// Functions/Keypoint Features/F_VN_FindReferenceKeyPointsInImageAKAZE

	{attribute 'TcIecLibraryType'}
	{attribute 'external_name' := 'F_VN_FindReferenceKeyPointsInImageAKAZE_GUID_B9801059_E7E5_45E6_F0CA_70766AD6A2AB'}
	(* Searches a reference image, represented by its AKAZE keypoints and corresponding descriptors, in a given source image (uses the default TcVnParamsAKAZE parameters). *)
	FUNCTION F_VN_FindReferenceKeyPointsInImageAKAZE : HRESULT
	VAR_INPUT
		ipSrcImage	:	ITcVnImage;	(* Source image *)
		ipRefKeyPoints	:	ITcVnContainer;	(* KeyPoints of the reference image, e.g. computed with F_VN_KeyPointsAndDescriptorsAKAZE (ContainerType_Vector_TcVnKeyPoint) *)
		ipRefDescriptors	:	ITcVnImage;	(* Descriptors of the reference image KeyPoints, e.g. computed with F_VN_KeyPointsAndDescriptorsAKAZE *)
		nRefImageWidth	:	UDINT;	(* Width of the reference image in pixels *)
		nRefImageHeight	:	UDINT;	(* Height of the reference image in pixels *)
		ipEdgePoints	:	REFERENCE TO ITcVnContainer;	(* Returns a container with the 4 edge points of the reference image transformed into ipSrcImage coordinates (ContainerType_Vector_TcVnPoint2_REAL) *)
		fMaxDist	:	REAL;	(* Maximum allowed descriptor distance (-1 disables this filter criterion) *)
		fMaxKnnRatio	:	REAL;	(* Maximum allowed distance ratio between first and second best match ([0..1], -1 disables this filter criterion) *)
		hrPrev	:	HRESULT;	(* HRESULT indicating the result of previous operations (If SUCCEEDED(hrPrev) equals false, no operation is executed.) *)
	END_VAR
	VAR_OUTPUT
		aPerspectiveTransform	:	TcVnMatrix3x3_LREAL;	(* Returns the perspective transformation matrix, which transforms the reference points to the source points *)
		nNumberOfGoodMatches	:	UDINT;	(* Return the number of good matches *)
		nNumberOfInliers	:	UDINT;	(* Return the number of inlier matches *)
	END_VAR

END_FUNCTION

// Functions/Keypoint Features/F_VN_KeyPointsAndDescriptorsAKAZE

	{attribute 'TcIecLibraryType'}
	{attribute 'external_name' := 'F_VN_KeyPointsAndDescriptorsAKAZE_GUID_33FCE752_CC73_4619_CE24_ACBC29908D23'}
	(* Detects keypoints and compute descriptors using the AKAZE method. *)
	FUNCTION F_VN_KeyPointsAndDescriptorsAKAZE : HRESULT
	VAR_INPUT
		ipSrcImage	:	ITcVnImage;	(* Source image *)
		ipKeyPoints	:	REFERENCE TO ITcVnContainer;	(* Returns a container which is filled with the keypoints (ContainerType_Vector_TcVnKeyPoint; Non-zero interface pointers are reused.) *)
		ipDescriptors	:	REFERENCE TO ITcVnImage;	(* Descriptor image (set to 0 if not required; 1 descriptor in each row; An appropriate image will be created if required.) *)
		hrPrev	:	HRESULT;	(* HRESULT indicating the result of previous operations (If SUCCEEDED(hrPrev) equals false, no operation is executed.) *)
	END_VAR

END_FUNCTION

// Functions/Keypoint Features/F_VN_FindReferenceKeyPointsInImageAKAZEExp

	{attribute 'TcIecLibraryType'}
	{attribute 'external_name' := 'F_VN_FindReferenceKeyPointsInImageAKAZEExp_GUID_5A20AA7D_A742_4EBE_E505_E1E5875E6765'}
	(* Searches a reference image, represented by its AKAZE keypoints and corresponding descriptors, in a given source image. (expert function) *)
	FUNCTION F_VN_FindReferenceKeyPointsInImageAKAZEExp : HRESULT
	VAR_INPUT
		ipSrcImage	:	ITcVnImage;	(* Source image *)
		ipRefKeyPoints	:	ITcVnContainer;	(* KeyPoints of the reference image, e.g. computed with F_VN_KeyPointsAndDescriptorsAKAZE (ContainerType_Vector_TcVnKeyPoint) *)
		ipRefDescriptors	:	ITcVnImage;	(* Descriptors of the reference image KeyPoints, e.g. computed with F_VN_KeyPointsAndDescriptorsAKAZE *)
		nRefImageWidth	:	UDINT;	(* Width of the reference image in pixels *)
		nRefImageHeight	:	UDINT;	(* Height of the reference image in pixels *)
		ipEdgePoints	:	REFERENCE TO ITcVnContainer;	(* Returns a container with the 4 edge points of the reference image transformed into ipSrcImage coordinates (ContainerType_Vector_TcVnPoint2_REAL) *)
		fMaxDist	:	REAL;	(* Maximum allowed descriptor distance (-1 disables this filter criterion) *)
		fMaxKnnRatio	:	REAL;	(* Maximum allowed distance ratio between first and second best match ([0..1], -1 disables this filter criterion) *)
		eNormType	:	ETcVnNormalizationType;	(* Normalization type used for descriptor matching *)
		ipSrcImageMask	:	ITcVnImage;	(* Mask to specify, where to look for keypoints in ipSrcImage (set to 0 if no mask required) *)
	END_VAR
	VAR_IN_OUT
		stAkazeParams	:	TcVnParamsAKAZE;	(* Parameters to configure the keypoint and descriptor computation for ipSrcImage (resulting descriptors must be compatible to ipRefDescriptors!) *)
	END_VAR
	VAR_INPUT
		eAlgorithm	:	ETcVnEstimationAlgorithm;	(* Estimation algorithm used for computing the perspective transformation between the two point sets *)
		fReprojThreshold	:	LREAL;	(* Maximum allowed reprojection error to treat a point pair as an inlier (only used if eAlgorithm is RANSAC, RHO) *)
		nMaxIterations	:	UDINT;	(* Maximum number of RANSAC iterations *)
		fConfidence	:	LREAL;	(* Confidence (0..1) *)
		hrPrev	:	HRESULT;	(* HRESULT indicating the result of previous operations (If SUCCEEDED(hrPrev) equals false, no operation is executed.) *)
	END_VAR
	VAR_OUTPUT
		aPerspectiveTransform	:	TcVnMatrix3x3_LREAL;	(* Returns the perspective transformation matrix, which transforms the reference points to the source points  *)
		nNumberOfGoodMatches	:	UDINT;	(* Return the number of good matches *)
		nNumberOfInliers	:	UDINT;	(* Return the number of inlier matches *)
	END_VAR

END_FUNCTION

// Functions/Keypoint Features/F_VN_FindReferenceKeyPointsInImageBRISK

	{attribute 'TcIecLibraryType'}
	{attribute 'external_name' := 'F_VN_FindReferenceKeyPointsInImageBRISK_GUID_C6B47D52_F5A1_4A13_CF78_EFB52692276F'}
	(* Searches a reference image, represented by its BRISK keypoints and corresponding descriptors, in a given source image (uses the default TcVnParamsBRISK parameters). *)
	FUNCTION F_VN_FindReferenceKeyPointsInImageBRISK : HRESULT
	VAR_INPUT
		ipSrcImage	:	ITcVnImage;	(* Source image *)
		ipRefKeyPoints	:	ITcVnContainer;	(* KeyPoints of the reference image, e.g. computed with F_VN_KeyPointsAndDescriptorsBRISK (ContainerType_Vector_TcVnKeyPoint) *)
		ipRefDescriptors	:	ITcVnImage;	(* Descriptors of the reference image KeyPoints, e.g. computed with F_VN_KeyPointsAndDescriptorsBRISK *)
		nRefImageWidth	:	UDINT;	(* Width of the reference image in pixels *)
		nRefImageHeight	:	UDINT;	(* Height of the reference image in pixels *)
		ipEdgePoints	:	REFERENCE TO ITcVnContainer;	(* Returns a container with the 4 edge points of the reference image transformed into ipSrcImage coordinates (ContainerType_Vector_TcVnPoint2_REAL) *)
		fMaxDist	:	REAL;	(* Maximum allowed descriptor distance (-1 disables this filter criterion) *)
		fMaxKnnRatio	:	REAL;	(* Maximum allowed distance ratio between first and second best match ([0..1], -1 disables this filter criterion) *)
		hrPrev	:	HRESULT;	(* HRESULT indicating the result of previous operations (If SUCCEEDED(hrPrev) equals false, no operation is executed.) *)
	END_VAR
	VAR_OUTPUT
		aPerspectiveTransform	:	TcVnMatrix3x3_LREAL;	(* Returns the perspective transformation matrix, which transforms the reference points to the source points  *)
		nNumberOfGoodMatches	:	UDINT;	(* Return the number of good matches *)
		nNumberOfInliers	:	UDINT;	(* Return the number of inlier matches *)
	END_VAR

END_FUNCTION

// Functions/Keypoint Features/F_VN_KeyPointsAndDescriptorsBRISK

	{attribute 'TcIecLibraryType'}
	{attribute 'external_name' := 'F_VN_KeyPointsAndDescriptorsBRISK_GUID_84C0A1DE_69BD_404B_FE31_2FE04FC65E23'}
	(* Detects keypoints and compute descriptors using the BRISK method. *)
	FUNCTION F_VN_KeyPointsAndDescriptorsBRISK : HRESULT
	VAR_INPUT
		ipSrcImage	:	ITcVnImage;	(* Source image *)
		ipKeyPoints	:	REFERENCE TO ITcVnContainer;	(* Returns a container which is filled with the keypoints (ContainerType_Vector_TcVnKeyPoint; Non-zero interface pointers are reused.) *)
		ipDescriptors	:	REFERENCE TO ITcVnImage;	(* Descriptor image (set to 0 if not required; 1 descriptor in each row; An appropriate image will be created if required.) *)
		hrPrev	:	HRESULT;	(* HRESULT indicating the result of previous operations (If SUCCEEDED(hrPrev) equals false, no operation is executed.) *)
	END_VAR

END_FUNCTION

// Functions/Keypoint Features/F_VN_FindReferenceKeyPointsInImageBRISKExp

	{attribute 'TcIecLibraryType'}
	{attribute 'external_name' := 'F_VN_FindReferenceKeyPointsInImageBRISKExp_GUID_84B8D030_BDDF_4ECF_E2AC_C4FA02ED163C'}
	(* Searches a reference image, represented by its BRISK keypoints and corresponding descriptors, in a given source image. (expert function) *)
	FUNCTION F_VN_FindReferenceKeyPointsInImageBRISKExp : HRESULT
	VAR_INPUT
		ipSrcImage	:	ITcVnImage;	(* Source image *)
		ipRefKeyPoints	:	ITcVnContainer;	(* KeyPoints of the reference image, e.g. computed with F_VN_KeyPointsAndDescriptorsBRISK (ContainerType_Vector_TcVnKeyPoint) *)
		ipRefDescriptors	:	ITcVnImage;	(* Descriptors of the reference image KeyPoints, e.g. computed with F_VN_KeyPointsAndDescriptorsBRISK *)
		nRefImageWidth	:	UDINT;	(* Width of the reference image in pixels *)
		nRefImageHeight	:	UDINT;	(* Height of the reference image in pixels *)
		ipEdgePoints	:	REFERENCE TO ITcVnContainer;	(* Returns a container with the 4 edge points of the reference image transformed into ipSrcImage coordinates (ContainerType_Vector_TcVnPoint2_REAL) *)
		fMaxDist	:	REAL;	(* Maximum allowed descriptor distance (-1 disables this filter criterion) *)
		fMaxKnnRatio	:	REAL;	(* Maximum allowed distance ratio between first and second best match ([0..1], -1 disables this filter criterion) *)
		eNormType	:	ETcVnNormalizationType;	(* Normalization type used for descriptor matching *)
		ipSrcImageMask	:	ITcVnImage;	(* Mask to specify, where to look for keypoints in ipSrcImage (set to 0 if no mask required) *)
	END_VAR
	VAR_IN_OUT
		stBriskParams	:	TcVnParamsBRISK;	(* Parameters to configure the keypoint and descriptor computation for ipSrcImage (resulting descriptors must be compatible to ipRefDescriptors!) *)
	END_VAR
	VAR_INPUT
		eAlgorithm	:	ETcVnEstimationAlgorithm;	(* Estimation algorithm used for computing the perspective transformation between the two point sets *)
		fReprojThreshold	:	LREAL;	(* Maximum allowed reprojection error to treat a point pair as an inlier (only used if eAlgorithm is RANSAC, RHO) *)
		nMaxIterations	:	UDINT;	(* Maximum number of RANSAC iterations *)
		fConfidence	:	LREAL;	(* Confidence (0..1) *)
		hrPrev	:	HRESULT;	(* HRESULT indicating the result of previous operations (If SUCCEEDED(hrPrev) equals false, no operation is executed.) *)
	END_VAR
	VAR_OUTPUT
		aPerspectiveTransform	:	TcVnMatrix3x3_LREAL;	(* Returns the perspective transformation matrix, which transforms the reference points to the source points  *)
		nNumberOfGoodMatches	:	UDINT;	(* Return the number of good matches *)
		nNumberOfInliers	:	UDINT;	(* Return the number of inlier matches *)
	END_VAR

END_FUNCTION

// Functions/Keypoint Features/F_VN_FindReferenceKeyPointsInImageORB

	{attribute 'TcIecLibraryType'}
	{attribute 'external_name' := 'F_VN_FindReferenceKeyPointsInImageORB_GUID_A7F5A2C2_C6E4_44AD_C84D_FFDC882441D3'}
	(* Searches a reference image, represented by its ORB keypoints and corresponding descriptors, in a given source image (uses the default TcVnParamsORB parameters). *)
	FUNCTION F_VN_FindReferenceKeyPointsInImageORB : HRESULT
	VAR_INPUT
		ipSrcImage	:	ITcVnImage;	(* Source image *)
		ipRefKeyPoints	:	ITcVnContainer;	(* KeyPoints of the reference image, e.g. computed with F_VN_KeyPointsAndDescriptorsORB (ContainerType_Vector_TcVnKeyPoint) *)
		ipRefDescriptors	:	ITcVnImage;	(* Descriptors of the reference image KeyPoints, e.g. computed with F_VN_KeyPointsAndDescriptorsORB *)
		nRefImageWidth	:	UDINT;	(* Width of the reference image in pixels *)
		nRefImageHeight	:	UDINT;	(* Height of the reference image in pixels *)
		ipEdgePoints	:	REFERENCE TO ITcVnContainer;	(* Returns a container with the 4 edge points of the reference image transformed into ipSrcImage coordinates (ContainerType_Vector_TcVnPoint2_REAL) *)
		fMaxDist	:	REAL;	(* Maximum allowed descriptor distance (-1 disables this filter criterion) *)
		fMaxKnnRatio	:	REAL;	(* Maximum allowed distance ratio between first and second best match ([0..1], -1 disables this filter criterion) *)
		hrPrev	:	HRESULT;	(* HRESULT indicating the result of previous operations (If SUCCEEDED(hrPrev) equals false, no operation is executed.) *)
	END_VAR
	VAR_OUTPUT
		aPerspectiveTransform	:	TcVnMatrix3x3_LREAL;	(* Returns the perspective transformation matrix, which transforms the reference points to the source points  *)
		nNumberOfGoodMatches	:	UDINT;	(* Return the number of good matches *)
		nNumberOfInliers	:	UDINT;	(* Return the number of inlier matches *)
	END_VAR

END_FUNCTION

// Functions/Keypoint Features/F_VN_KeyPointsAndDescriptorsORB

	{attribute 'TcIecLibraryType'}
	{attribute 'external_name' := 'F_VN_KeyPointsAndDescriptorsORB_GUID_9F56F5E3_A789_412C_FE23_0DB22E24DDFB'}
	(* Detects keypoints and compute descriptors using the ORB method. *)
	FUNCTION F_VN_KeyPointsAndDescriptorsORB : HRESULT
	VAR_INPUT
		ipSrcImage	:	ITcVnImage;	(* Source image *)
		ipKeyPoints	:	REFERENCE TO ITcVnContainer;	(* Returns a container which is filled with the keypoints (ContainerType_Vector_TcVnKeyPoint; Non-zero interface pointers are reused.) *)
		ipDescriptors	:	REFERENCE TO ITcVnImage;	(* Descriptor image (set to 0 if not required; 1 descriptor in each row; An appropriate image will be created if required.) *)
		hrPrev	:	HRESULT;	(* HRESULT indicating the result of previous operations (If SUCCEEDED(hrPrev) equals false, no operation is executed.) *)
	END_VAR

END_FUNCTION

// Functions/Keypoint Features/F_VN_FindReferenceKeyPointsInImageORBExp

	{attribute 'TcIecLibraryType'}
	{attribute 'external_name' := 'F_VN_FindReferenceKeyPointsInImageORBExp_GUID_7AF107AB_9CF8_4ECC_CBE6_E3CD3540C632'}
	(* Searches a reference image, represented by its ORB keypoints and corresponding descriptors, in a given source image. (expert function) *)
	FUNCTION F_VN_FindReferenceKeyPointsInImageORBExp : HRESULT
	VAR_INPUT
		ipSrcImage	:	ITcVnImage;	(* Source image *)
		ipRefKeyPoints	:	ITcVnContainer;	(* KeyPoints of the reference image, e.g. computed with F_VN_KeyPointsAndDescriptorsORB (ContainerType_Vector_TcVnKeyPoint) *)
		ipRefDescriptors	:	ITcVnImage;	(* Descriptors of the reference image KeyPoints, e.g. computed with F_VN_KeyPointsAndDescriptorsORB *)
		nRefImageWidth	:	UDINT;	(* Width of the reference image in pixels *)
		nRefImageHeight	:	UDINT;	(* Height of the reference image in pixels *)
		ipEdgePoints	:	REFERENCE TO ITcVnContainer;	(* Returns a container with the 4 edge points of the reference image transformed into ipSrcImage coordinates (ContainerType_Vector_TcVnPoint2_REAL) *)
		fMaxDist	:	REAL;	(* Maximum allowed descriptor distance (-1 disables this filter criterion) *)
		fMaxKnnRatio	:	REAL;	(* Maximum allowed distance ratio between first and second best match ([0..1], -1 disables this filter criterion) *)
		eNormType	:	ETcVnNormalizationType;	(* Normalization type used for descriptor matching (HAMMING recommended for ORB, HAMMING2 if the ORB nBriefPoints parameter is 3 or 4) *)
		ipSrcImageMask	:	ITcVnImage;	(* Mask to specify, where to look for keypoints in ipSrcImage (set to 0 if no mask required) *)
	END_VAR
	VAR_IN_OUT
		stOrbParams	:	TcVnParamsORB;	(* Parameters to configure the keypoint and descriptor computation for ipSrcImage (resulting descriptors must be compatible to ipRefDescriptors!) *)
	END_VAR
	VAR_INPUT
		eAlgorithm	:	ETcVnEstimationAlgorithm;	(* Estimation algorithm used for computing the perspective transformation between the two point sets *)
		fReprojThreshold	:	LREAL;	(* Maximum allowed reprojection error to treat a point pair as an inlier (only used if eAlgorithm is RANSAC, RHO) *)
		nMaxIterations	:	UDINT;	(* Maximum number of RANSAC iterations *)
		fConfidence	:	LREAL;	(* Confidence (0..1) *)
		hrPrev	:	HRESULT;	(* HRESULT indicating the result of previous operations (If SUCCEEDED(hrPrev) equals false, no operation is executed.) *)
	END_VAR
	VAR_OUTPUT
		aPerspectiveTransform	:	TcVnMatrix3x3_LREAL;	(* Returns the perspective transformation matrix, which transforms the reference points to the source points  *)
		nNumberOfGoodMatches	:	UDINT;	(* Return the number of good matches *)
		nNumberOfInliers	:	UDINT;	(* Return the number of inlier matches *)
	END_VAR

END_FUNCTION

// Functions/Keypoint Features/F_VN_GetMatchCoordinates

	{attribute 'TcIecLibraryType'}
	{attribute 'external_name' := 'F_VN_GetMatchCoordinates_GUID_C88C0A54_949E_49E1_C497_E5D2AD49D6C8'}
	(* Return the coordinates of keypoints that match each other. *)
	FUNCTION F_VN_GetMatchCoordinates : HRESULT
	VAR_INPUT
		ipQueryKeyPoints	:	ITcVnContainer;	(* Container with query Keypoints (i.e. keypoints of a reference/template image) of type CTcVnContainer_Vector_TcVnKeyPoint *)
		ipTrainKeyPoints	:	ITcVnContainer;	(* Container with training Keypoints (i.e. keypoints of a source/input image) of type CTcVnContainer_Vector_TcVnKeyPoint *)
		ipMatches	:	ITcVnContainer;	(* Container with matches between query and train Keypoints (CTcVnContainer_Vector_TcVnDMatch). *)
		ipQueryCoordinates	:	REFERENCE TO ITcVnContainer;	(* Returns a container with the coordinates of keypoints from the query Keypoints that exist in ipMatches (CTcVnContainer_Vector_TcVnPoint2_REAL) *)
		ipTrainCoordinates	:	REFERENCE TO ITcVnContainer;	(* Returns a container with the coordinates of keypoints from the training Keypoints that exist in ipMatches (CTcVnContainer_Vector_TcVnPoint2_REAL) *)
		hrPrev	:	HRESULT;	(* HRESULT indicating the result of previous operations (If SUCCEEDED(hrPrev) equals false, no operation is executed.) *)
	END_VAR

END_FUNCTION

// Functions/Keypoint Features/F_VN_KeyPointsAGAST

	{attribute 'TcIecLibraryType'}
	{attribute 'external_name' := 'F_VN_KeyPointsAGAST_GUID_8B1DD5EA_B426_4523_FF3F_46B91ECE4C11'}
	(* Detects keypoints using the AGAST method. *)
	FUNCTION F_VN_KeyPointsAGAST : HRESULT
	VAR_INPUT
		ipSrcImage	:	ITcVnImage;	(* Source image *)
		ipKeyPoints	:	REFERENCE TO ITcVnContainer;	(* Returns a container which is filled with the keypoints (ContainerType_Vector_TcVnKeyPoint; Non-zero interface pointers are reused.) *)
		hrPrev	:	HRESULT;	(* HRESULT indicating the result of previous operations (If SUCCEEDED(hrPrev) equals false, no operation is executed.) *)
	END_VAR

END_FUNCTION

// Functions/Keypoint Features/F_VN_KeyPointsAGASTExp

	{attribute 'TcIecLibraryType'}
	{attribute 'external_name' := 'F_VN_KeyPointsAGASTExp_GUID_9C6794C7_3BEF_4308_C500_CB20EAF4E87E'}
	(* Detects keypoints using the AGAST method. (expert function) *)
	FUNCTION F_VN_KeyPointsAGASTExp : HRESULT
	VAR_INPUT
		ipSrcImage	:	ITcVnImage;	(* Source image *)
		ipKeyPoints	:	REFERENCE TO ITcVnContainer;	(* Returns a container which is filled with the keypoints (ContainerType_Vector_TcVnKeyPoint; Non-zero interface pointers are reused.) *)
		ipMask	:	ITcVnImage;	(* Mask to specify, where to look for keypoints (set to 0 if no mask required) *)
	END_VAR
	VAR_IN_OUT
		stParams	:	TcVnParamsAGAST;	(* Additional expert parameters *)
	END_VAR
	VAR_INPUT
		hrPrev	:	HRESULT;	(* HRESULT indicating the result of previous operations (If SUCCEEDED(hrPrev) equals false, no operation is executed.) *)
	END_VAR

END_FUNCTION

// Functions/Keypoint Features/F_VN_KeyPointsAndDescriptorsAKAZEExp

	{attribute 'TcIecLibraryType'}
	{attribute 'external_name' := 'F_VN_KeyPointsAndDescriptorsAKAZEExp_GUID_6BF621AA_B810_4C4A_F2A0_C697F464C22F'}
	(* Detects keypoints and compute descriptors using the AKAZE method. (expert function) *)
	FUNCTION F_VN_KeyPointsAndDescriptorsAKAZEExp : HRESULT
	VAR_INPUT
		ipSrcImage	:	ITcVnImage;	(* Source image *)
		ipKeyPoints	:	REFERENCE TO ITcVnContainer;	(* Returns a container which is filled with the keypoints (ContainerType_Vector_TcVnKeyPoint; Non-zero interface pointers are reused.) *)
		ipDescriptors	:	REFERENCE TO ITcVnImage;	(* Descriptor image (set to 0 if not required; 1 descriptor in each row; An appropriate image will be created if required.) *)
		ipMask	:	ITcVnImage;	(* Mask to specify, where to look for keypoints (set to 0 if no mask required) *)
	END_VAR
	VAR_IN_OUT
		stParams	:	TcVnParamsAKAZE;	(* Additional expert parameters *)
	END_VAR
	VAR_INPUT
		hrPrev	:	HRESULT;	(* HRESULT indicating the result of previous operations (If SUCCEEDED(hrPrev) equals false, no operation is executed.) *)
	END_VAR

END_FUNCTION

// Functions/Keypoint Features/F_VN_KeyPointsAndDescriptorsBRISKExp

	{attribute 'TcIecLibraryType'}
	{attribute 'external_name' := 'F_VN_KeyPointsAndDescriptorsBRISKExp_GUID_DA6DD11F_0B80_47B6_D05E_C63065A602A3'}
	(* Detects keypoints and compute descriptors using the BRISK method. (expert function) *)
	FUNCTION F_VN_KeyPointsAndDescriptorsBRISKExp : HRESULT
	VAR_INPUT
		ipSrcImage	:	ITcVnImage;	(* Source image *)
		ipKeyPoints	:	REFERENCE TO ITcVnContainer;	(* Returns a container which is filled with the keypoints (ContainerType_Vector_TcVnKeyPoint; Non-zero interface pointers are reused.) *)
		ipDescriptors	:	REFERENCE TO ITcVnImage;	(* Descriptor image (set to 0 if not required; 1 descriptor in each row; An appropriate image will be created if required.) *)
		ipMask	:	ITcVnImage;	(* Mask to specify, where to look for keypoints (set to 0 if no mask required) *)
	END_VAR
	VAR_IN_OUT
		stParams	:	TcVnParamsBRISK;	(* Additional expert parameters *)
	END_VAR
	VAR_INPUT
		hrPrev	:	HRESULT;	(* HRESULT indicating the result of previous operations (If SUCCEEDED(hrPrev) equals false, no operation is executed.) *)
	END_VAR

END_FUNCTION

// Functions/Keypoint Features/F_VN_KeyPointsAndDescriptorsKAZE

	{attribute 'TcIecLibraryType'}
	{attribute 'external_name' := 'F_VN_KeyPointsAndDescriptorsKAZE_GUID_CB7E23FD_64FC_4AB3_CD2C_813AD0BC8653'}
	(* Detects keypoints and compute descriptors using the KAZE method. *)
	FUNCTION F_VN_KeyPointsAndDescriptorsKAZE : HRESULT
	VAR_INPUT
		ipSrcImage	:	ITcVnImage;	(* Source image *)
		ipKeyPoints	:	REFERENCE TO ITcVnContainer;	(* Returns a container which is filled with the keypoints (ContainerType_Vector_TcVnKeyPoint; Non-zero interface pointers are reused.) *)
		ipDescriptors	:	REFERENCE TO ITcVnImage;	(* Descriptor image (set to 0 if not required; 1 descriptor in each row; An appropriate image will be created if required.) *)
		hrPrev	:	HRESULT;	(* HRESULT indicating the result of previous operations (If SUCCEEDED(hrPrev) equals false, no operation is executed.) *)
	END_VAR

END_FUNCTION

// Functions/Keypoint Features/F_VN_KeyPointsAndDescriptorsKAZEExp

	{attribute 'TcIecLibraryType'}
	{attribute 'external_name' := 'F_VN_KeyPointsAndDescriptorsKAZEExp_GUID_ABCD74A9_0266_46D0_DE82_C1B896FFC393'}
	(* Detects keypoints and compute descriptors using the KAZE method. (expert function) *)
	FUNCTION F_VN_KeyPointsAndDescriptorsKAZEExp : HRESULT
	VAR_INPUT
		ipSrcImage	:	ITcVnImage;	(* Source image *)
		ipKeyPoints	:	REFERENCE TO ITcVnContainer;	(* Returns a container which is filled with the keypoints (ContainerType_Vector_TcVnKeyPoint; Non-zero interface pointers are reused.) *)
		ipDescriptors	:	REFERENCE TO ITcVnImage;	(* Descriptor image (set to 0 if not required; 1 descriptor in each row; An appropriate image will be created if required.) *)
		ipMask	:	ITcVnImage;	(* Mask to specify, where to look for keypoints (set to 0 if no mask required) *)
	END_VAR
	VAR_IN_OUT
		stParams	:	TcVnParamsKAZE;	(* Additional expert parameters *)
	END_VAR
	VAR_INPUT
		hrPrev	:	HRESULT;	(* HRESULT indicating the result of previous operations (If SUCCEEDED(hrPrev) equals false, no operation is executed.) *)
	END_VAR

END_FUNCTION

// Functions/Keypoint Features/F_VN_KeyPointsAndDescriptorsORBExp

	{attribute 'TcIecLibraryType'}
	{attribute 'external_name' := 'F_VN_KeyPointsAndDescriptorsORBExp_GUID_E2CE0C5B_D279_493E_DF06_AF7BB41166C3'}
	(* Detect keypoints and compute descriptors using the ORB method. (expert function) *)
	FUNCTION F_VN_KeyPointsAndDescriptorsORBExp : HRESULT
	VAR_INPUT
		ipSrcImage	:	ITcVnImage;	(* Source image *)
		ipKeyPoints	:	REFERENCE TO ITcVnContainer;	(* Returns a container which is filled with the keypoints (ContainerType_Vector_TcVnKeyPoint; Non-zero interface pointers are reused.) *)
		ipDescriptors	:	REFERENCE TO ITcVnImage;	(* Descriptor image (set to 0 if not required; 1 descriptor in each row; An appropriate image will be created if required.) *)
		ipMask	:	ITcVnImage;	(* Mask to specify, where to look for keypoints (set to 0 if no mask required) *)
	END_VAR
	VAR_IN_OUT
		stParams	:	TcVnParamsORB;	(* Additional expert parameters *)
	END_VAR
	VAR_INPUT
		hrPrev	:	HRESULT;	(* HRESULT indicating the result of previous operations (If SUCCEEDED(hrPrev) equals false, no operation is executed.) *)
	END_VAR

END_FUNCTION

// Functions/Keypoint Features/F_VN_KeyPointsFAST

	{attribute 'TcIecLibraryType'}
	{attribute 'external_name' := 'F_VN_KeyPointsFAST_GUID_53C69CE8_4FD7_49A4_F786_656C1415DC0F'}
	(* Detects keypoints using the FAST method. *)
	FUNCTION F_VN_KeyPointsFAST : HRESULT
	VAR_INPUT
		ipSrcImage	:	ITcVnImage;	(* Source image (single-channel). *)
		ipKeyPoints	:	REFERENCE TO ITcVnContainer;	(* Returns a container which is filled with the keypoints (ContainerType_Vector_TcVnKeyPoint; Non-zero interface pointers are reused.) *)
		hrPrev	:	HRESULT;	(* HRESULT indicating the result of previous operations (If SUCCEEDED(hrPrev) equals false, no operation is executed.) *)
	END_VAR

END_FUNCTION

// Functions/Keypoint Features/F_VN_KeyPointsFASTExp

	{attribute 'TcIecLibraryType'}
	{attribute 'external_name' := 'F_VN_KeyPointsFASTExp_GUID_891C3F83_599D_4E10_E84A_099C436BFDFA'}
	(* Detects keypoints using the FAST method. (expert function) *)
	FUNCTION F_VN_KeyPointsFASTExp : HRESULT
	VAR_INPUT
		ipSrcImage	:	ITcVnImage;	(* Source image *)
		ipKeyPoints	:	REFERENCE TO ITcVnContainer;	(* Returns a container which is filled with the keypoints (ContainerType_Vector_TcVnKeyPoint; Non-zero interface pointers are reused.) *)
		ipMask	:	ITcVnImage;	(* Mask to specify, where to look for keypoints (set to 0 if no mask required) *)
	END_VAR
	VAR_IN_OUT
		stParams	:	TcVnParamsFAST;	(* Additional expert parameters *)
	END_VAR
	VAR_INPUT
		hrPrev	:	HRESULT;	(* HRESULT indicating the result of previous operations (If SUCCEEDED(hrPrev) equals false, no operation is executed.) *)
	END_VAR

END_FUNCTION

// Functions/Keypoint Features/F_VN_KeyPointsGFTT

	{attribute 'TcIecLibraryType'}
	{attribute 'external_name' := 'F_VN_KeyPointsGFTT_GUID_4B437876_D85E_4CC7_C916_7160C7C18A8B'}
	(* Detects keypoints using the GFTT method, which detects strong corners. *)
	FUNCTION F_VN_KeyPointsGFTT : HRESULT
	VAR_INPUT
		ipSrcImage	:	ITcVnImage;	(* Source image *)
		ipKeyPoints	:	REFERENCE TO ITcVnContainer;	(* Returns a container which is filled with the keypoints (ContainerType_Vector_TcVnKeyPoint; Non-zero interface pointers are reused.) *)
		hrPrev	:	HRESULT;	(* HRESULT indicating the result of previous operations (If SUCCEEDED(hrPrev) equals false, no operation is executed.) *)
	END_VAR

END_FUNCTION

// Functions/Keypoint Features/F_VN_KeyPointsGFTTExp

	{attribute 'TcIecLibraryType'}
	{attribute 'external_name' := 'F_VN_KeyPointsGFTTExp_GUID_C73D6DBE_2B80_4E2D_D1B9_0989E68A55CA'}
	(* Detects keypoints using the GFTT method, which detects strong corners. (expert function) *)
	FUNCTION F_VN_KeyPointsGFTTExp : HRESULT
	VAR_INPUT
		ipSrcImage	:	ITcVnImage;	(* Source image *)
		ipKeyPoints	:	REFERENCE TO ITcVnContainer;	(* Returns a container which is filled with the keypoints (ContainerType_Vector_TcVnKeyPoint; Non-zero interface pointers are reused.) *)
		ipMask	:	ITcVnImage;	(* Mask to specify, where to look for keypoints (set to 0 if no mask required) *)
	END_VAR
	VAR_IN_OUT
		stParams	:	TcVnParamsGFTT;	(* Additional expert parameters *)
	END_VAR
	VAR_INPUT
		hrPrev	:	HRESULT;	(* HRESULT indicating the result of previous operations (If SUCCEEDED(hrPrev) equals false, no operation is executed.) *)
	END_VAR

END_FUNCTION

// Functions/Keypoint Features/F_VN_KeyPointsMSER

	{attribute 'TcIecLibraryType'}
	{attribute 'external_name' := 'F_VN_KeyPointsMSER_GUID_35659FE7_48EA_4456_C1E0_923144E2D01C'}
	(* Detects keypoints using the MSER method. *)
	FUNCTION F_VN_KeyPointsMSER : HRESULT
	VAR_INPUT
		ipSrcImage	:	ITcVnImage;	(* Source image *)
		ipKeyPoints	:	REFERENCE TO ITcVnContainer;	(* Returns a container which is filled with the keypoints (ContainerType_Vector_TcVnKeyPoint; Non-zero interface pointers are reused.) *)
		hrPrev	:	HRESULT;	(* HRESULT indicating the result of previous operations (If SUCCEEDED(hrPrev) equals false, no operation is executed.) *)
	END_VAR

END_FUNCTION

// Functions/Keypoint Features/F_VN_KeyPointsMSERExp

	{attribute 'TcIecLibraryType'}
	{attribute 'external_name' := 'F_VN_KeyPointsMSERExp_GUID_C7BACDB3_FAB3_4B5C_F885_22F0A9028035'}
	(* Detects keypoints using the MSER method. (expert function) *)
	FUNCTION F_VN_KeyPointsMSERExp : HRESULT
	VAR_INPUT
		ipSrcImage	:	ITcVnImage;	(* Source image *)
		ipKeyPoints	:	REFERENCE TO ITcVnContainer;	(* Returns a container which is filled with the keypoints (ContainerType_Vector_TcVnKeyPoint; Non-zero interface pointers are reused.) *)
		ipMask	:	ITcVnImage;	(* Mask to specify, where to look for keypoints (set to 0 if no mask required) *)
	END_VAR
	VAR_IN_OUT
		stParams	:	TcVnParamsMSER;	(* Additional expert parameters *)
	END_VAR
	VAR_INPUT
		hrPrev	:	HRESULT;	(* HRESULT indicating the result of previous operations (If SUCCEEDED(hrPrev) equals false, no operation is executed.) *)
	END_VAR

END_FUNCTION

// Functions/Keypoint Features/F_VN_KeyPointsSB

	{attribute 'TcIecLibraryType'}
	{attribute 'external_name' := 'F_VN_KeyPointsSB_GUID_46A8286A_E09D_435E_E1F3_2458A1D98CFC'}
	(* Detects keypoints using a Simple Blob method
          - several iterations apply different thresholds to source image
          - connected components (blobs) are detected
          - the center and radius of the blobs are returned as keypoints *)
	FUNCTION F_VN_KeyPointsSB : HRESULT
	VAR_INPUT
		ipSrcImage	:	ITcVnImage;	(* Source image *)
		ipKeyPoints	:	REFERENCE TO ITcVnContainer;	(* Returns a container which is filled with the keypoints (ContainerType_Vector_TcVnKeyPoint; Non-zero interface pointers are reused.) *)
		hrPrev	:	HRESULT;	(* HRESULT indicating the result of previous operations (If SUCCEEDED(hrPrev) equals false, no operation is executed.) *)
	END_VAR

END_FUNCTION

// Functions/Keypoint Features/F_VN_KeyPointsSBExp

	{attribute 'TcIecLibraryType'}
	{attribute 'external_name' := 'F_VN_KeyPointsSBExp_GUID_EDAC9E5C_09B7_4A6F_F6F2_EEC9A5D3E62F'}
	(* Detects keypoints using a Simple Blob method (expert function)
          - several iterations apply different thresholds to source image
          - connected components (blobs) are detected
          - the center and radius of the blobs are returned as keypoints *)
	FUNCTION F_VN_KeyPointsSBExp : HRESULT
	VAR_INPUT
		ipSrcImage	:	ITcVnImage;	(* Source image *)
		ipKeyPoints	:	REFERENCE TO ITcVnContainer;	(* Returns a container which is filled with the keypoints (ContainerType_Vector_TcVnKeyPoint; Non-zero interface pointers are reused.) *)
		ipMask	:	ITcVnImage;	(* Mask to specify, where to look for keypoints (optional, set to 0 if not required) *)
	END_VAR
	VAR_IN_OUT
		stParams	:	TcVnParamsSB;	(* Several parameters to filter the detected blobs *)
	END_VAR
	VAR_INPUT
		hrPrev	:	HRESULT;	(* HRESULT indicating the result of previous operations (If SUCCEEDED(hrPrev) equals false, no operation is executed.) *)
	END_VAR

END_FUNCTION

// Functions/Keypoint Features/F_VN_MatchDescriptorsBF

	{attribute 'TcIecLibraryType'}
	{attribute 'external_name' := 'F_VN_MatchDescriptorsBF_GUID_DFCE8028_706D_4AAE_ED57_9BEEBBC16700'}
	(* Match descriptors using a brute force approach. *)
	FUNCTION F_VN_MatchDescriptorsBF : HRESULT
	VAR_INPUT
		ipQueryDescriptors	:	ITcVnImage;	(* Query descriptors (i.e. descriptors of a reference/template image) *)
		ipTrainDescriptors	:	ITcVnImage;	(* Training descriptors (i.e. descriptors of a source/input image) *)
		ipMatches	:	REFERENCE TO ITcVnContainer;	(* Returns a container which is filled with the descriptor matches (ContainerType_Vector_TcVnDMatch; Non-zero interface pointers are reused.) *)
		hrPrev	:	HRESULT;	(* HRESULT indicating the result of previous operations (If SUCCEEDED(hrPrev) equals false, no operation is executed.) *)
	END_VAR

END_FUNCTION

// Functions/Keypoint Features/F_VN_MatchDescriptorsBFExp

	{attribute 'TcIecLibraryType'}
	{attribute 'external_name' := 'F_VN_MatchDescriptorsBFExp_GUID_2EDBDB49_F422_4007_D6F4_A3B58EEA9B1C'}
	(* Match descriptors using a brute force approach. (expert function) *)
	FUNCTION F_VN_MatchDescriptorsBFExp : HRESULT
	VAR_INPUT
		ipQueryDescriptors	:	ITcVnImage;	(* Query descriptors (i.e. descriptors of a reference/template image) *)
		ipTrainDescriptors	:	ITcVnImage;	(* Training descriptors (i.e. descriptors of a source/input image) *)
		ipMatches	:	REFERENCE TO ITcVnContainer;	(* Returns a container which is filled with the descriptor matches (ContainerType_Vector_TcVnDMatch; Non-zero interface pointers are reused.) *)
		ipMask	:	ITcVnImage;	(* Mask to specify permissable matches, i.e. query[i] can be matched with train[j] only if mask[i][j] != 0 (set to 0 if no mask required) *)
		eNormType	:	ETcVnNormalizationType;	(* Normalization type (only L1, L2, L2SQR, HAMMING, HAMMING2 supported). HAMMING2 should be used for ORB descriptors if the ORB nBriefPoints parameter is 3 or 4) *)
		bCrossCheck	:	BOOL;	(* If true, only consistent matches are returned, i.e. query->train and train->query detect the same match *)
		hrPrev	:	HRESULT;	(* HRESULT indicating the result of previous operations (If SUCCEEDED(hrPrev) equals false, no operation is executed.) *)
	END_VAR

END_FUNCTION

// Functions/Keypoint Features/F_VN_MatchDescriptorsFlannLsh

	{attribute 'TcIecLibraryType'}
	{attribute 'external_name' := 'F_VN_MatchDescriptorsFlannLsh_GUID_0650836A_7665_4286_CDF9_EFAAFCD2456E'}
	(* Match descriptors using a FLANN based approach with LSH index. *)
	FUNCTION F_VN_MatchDescriptorsFlannLsh : HRESULT
	VAR_INPUT
		ipQueryDescriptors	:	ITcVnImage;	(* Query descriptors (i.e. descriptors of a reference/template image) *)
		ipTrainDescriptors	:	ITcVnImage;	(* Training descriptors (i.e. descriptors of a source/input image) *)
		ipMatches	:	REFERENCE TO ITcVnContainer;	(* Returns a container which is filled with the descriptor matches (ContainerType_Vector_TcVnDMatch; Non-zero interface pointers are reused.) *)
		hrPrev	:	HRESULT;	(* HRESULT indicating the result of previous operations (If SUCCEEDED(hrPrev) equals false, no operation is executed.) *)
	END_VAR

END_FUNCTION

// Functions/Keypoint Features/F_VN_MatchDescriptorsFlannLshExp

	{attribute 'TcIecLibraryType'}
	{attribute 'external_name' := 'F_VN_MatchDescriptorsFlannLshExp_GUID_CAEC8F2F_95FF_436B_DA1E_847948374BE5'}
	(* Match descriptors using a FLANN based approach with LSH index. (expert function) *)
	FUNCTION F_VN_MatchDescriptorsFlannLshExp : HRESULT
	VAR_INPUT
		ipQueryDescriptors	:	ITcVnImage;	(* Query descriptors (i.e. descriptors of a reference/template image) *)
		ipTrainDescriptors	:	ITcVnImage;	(* Training descriptors (i.e. descriptors of a source/input image) *)
		ipMatches	:	REFERENCE TO ITcVnContainer;	(* Returns a container which is filled with the descriptor matches (ContainerType_Vector_TcVnDMatch; Non-zero interface pointers are reused.) *)
		nTableNumber	:	UDINT;	(* Number of tables *)
		nKeySize	:	UDINT;	(* Key size *)
		nMultiProbeLevel	:	UDINT;	(* Multi-probe level *)
		nChecks	:	UDINT;	(* Maximum number of visited leafs when searching for neighbors *)
		hrPrev	:	HRESULT;	(* HRESULT indicating the result of previous operations (If SUCCEEDED(hrPrev) equals false, no operation is executed.) *)
	END_VAR

END_FUNCTION

// Functions/Keypoint Features/F_VN_MatchDescriptorsKnnBF

	{attribute 'TcIecLibraryType'}
	{attribute 'external_name' := 'F_VN_MatchDescriptorsKnnBF_GUID_6F70A548_605A_4D10_E5BC_BB269C95F284'}
	(* Match descriptors (k nearest neighbors) using a brute force approach. *)
	FUNCTION F_VN_MatchDescriptorsKnnBF : HRESULT
	VAR_INPUT
		ipQueryDescriptors	:	ITcVnImage;	(* Query descriptors (i.e. descriptors of a reference/template image) *)
		ipTrainDescriptors	:	ITcVnImage;	(* Training descriptors (i.e. descriptors of a source/input image) *)
		ipMatches	:	REFERENCE TO ITcVnContainer;	(* Returns a container which is filled with the descriptor matches (ContainerType_Vector_Vector_TcVnDMatch; Non-zero interface pointers are reused.) *)
		nK	:	UDINT;	(* Number of required best train matches for each query descriptor (i.e. nk := 2) *)
		hrPrev	:	HRESULT;	(* HRESULT indicating the result of previous operations (If SUCCEEDED(hrPrev) equals false, no operation is executed.) *)
	END_VAR

END_FUNCTION

// Functions/Keypoint Features/F_VN_MatchDescriptorsKnnBFExp

	{attribute 'TcIecLibraryType'}
	{attribute 'external_name' := 'F_VN_MatchDescriptorsKnnBFExp_GUID_2307A43C_86AC_4610_DD2F_023DAB2AC390'}
	(* Match descriptors (k nearest neighbors) using a brute force approach. (expert function) *)
	FUNCTION F_VN_MatchDescriptorsKnnBFExp : HRESULT
	VAR_INPUT
		ipQueryDescriptors	:	ITcVnImage;	(* Query descriptors (i.e. descriptors of a reference/template image) *)
		ipTrainDescriptors	:	ITcVnImage;	(* Training descriptors (i.e. descriptors of a source/input image) *)
		ipMatches	:	REFERENCE TO ITcVnContainer;	(* Returns a container which is filled with the descriptor matches (ContainerType_Vector_Vector_TcVnDMatch; Non-zero interface pointers are reused.) *)
		nK	:	UDINT;	(* Number of required best train matches for each query descriptor (i.e. nk := 2) *)
		ipMask	:	ITcVnImage;	(* Mask to specify permissable matches, i.e. query[i] can be matched with train[j] only if mask[i][j] != 0 (set to 0 if no mask required) *)
		bCompactResult	:	BOOL;	(* If true, matches vector does not contain entries for fully masked-out query descriptors *)
		eNormType	:	ETcVnNormalizationType;	(* Normalization type (only L1, L2, L2SQR, HAMMING, HAMMING2 supported). HAMMING2 should be used for ORB descriptors if the ORB nBriefPoints parameter is 3 or 4) *)
		bCrossCheck	:	BOOL;	(* If true, only consistent matches are returned, i.e. query->train and train->query detect the same match (only used if nK = 1) *)
		hrPrev	:	HRESULT;	(* HRESULT indicating the result of previous operations (If SUCCEEDED(hrPrev) equals false, no operation is executed.) *)
	END_VAR

END_FUNCTION

// Functions/Keypoint Features/F_VN_MatchDescriptorsKnnFlannLsh

	{attribute 'TcIecLibraryType'}
	{attribute 'external_name' := 'F_VN_MatchDescriptorsKnnFlannLsh_GUID_A47CA1DA_0FA6_4D61_EB95_8BB5E9740C0B'}
	(* Match descriptors (k nearest neighbors) using a FLANN based approach with LSH index. *)
	FUNCTION F_VN_MatchDescriptorsKnnFlannLsh : HRESULT
	VAR_INPUT
		ipQueryDescriptors	:	ITcVnImage;	(* Query descriptors (i.e. descriptors of a reference/template image) *)
		ipTrainDescriptors	:	ITcVnImage;	(* Training descriptors (i.e. descriptors of a source/input image) *)
		ipMatches	:	REFERENCE TO ITcVnContainer;	(* Returns a container which is filled with the descriptor matches (ContainerType_Vector_Vector_TcVnDMatch; Non-zero interface pointers are reused.) *)
		nK	:	UDINT;	(* Number of required best train matches for each query descriptor (i.e. nk := 2) *)
		hrPrev	:	HRESULT;	(* HRESULT indicating the result of previous operations (If SUCCEEDED(hrPrev) equals false, no operation is executed.) *)
	END_VAR

END_FUNCTION

// Functions/Keypoint Features/F_VN_MatchDescriptorsKnnFlannLshExp

	{attribute 'TcIecLibraryType'}
	{attribute 'external_name' := 'F_VN_MatchDescriptorsKnnFlannLshExp_GUID_A8C4F9E1_4424_4D00_F6C1_9EE96948DA53'}
	(* Match descriptors (k nearest neighbors) using a FLANN based approach with LSH index. (expert function) *)
	FUNCTION F_VN_MatchDescriptorsKnnFlannLshExp : HRESULT
	VAR_INPUT
		ipQueryDescriptors	:	ITcVnImage;	(* Query descriptors (i.e. descriptors of a reference/template image) *)
		ipTrainDescriptors	:	ITcVnImage;	(* Training descriptors (i.e. descriptors of a source/input image) *)
		ipMatches	:	REFERENCE TO ITcVnContainer;	(* Returns a container which is filled with the descriptor matches (ContainerType_Vector_Vector_TcVnDMatch; Non-zero interface pointers are reused.) *)
		nK	:	UDINT;	(* Number of required best train matches for each query descriptor (i.e. nk := 2) *)
		nTableNumber	:	UDINT;	(* Number of tables *)
		nKeySize	:	UDINT;	(* Key size *)
		nMultiProbeLevel	:	UDINT;	(* Multi-probe level *)
		nChecks	:	UDINT;	(* Maximum number of visited leafs when searching for neighbors *)
		hrPrev	:	HRESULT;	(* HRESULT indicating the result of previous operations (If SUCCEEDED(hrPrev) equals false, no operation is executed.) *)
	END_VAR

END_FUNCTION

// Functions/Keypoint Features/F_VN_RegionsMSER

	{attribute 'TcIecLibraryType'}
	{attribute 'external_name' := 'F_VN_RegionsMSER_GUID_392CFCEB_3BBB_4D21_F20A_5BECED694B84'}
	(* Detects regions using the MSER method. *)
	FUNCTION F_VN_RegionsMSER : HRESULT
	VAR_INPUT
		ipSrcImage	:	ITcVnImage;	(* Source image *)
		ipRegions	:	REFERENCE TO ITcVnContainer;	(* Returns a container which is filled with the region points (ContainerType_Vector_Vector_TcVnPoint2_DINT; Non-zero interface pointers are reused.) *)
		ipBoundingBoxes	:	REFERENCE TO ITcVnContainer;	(* Returns a container which is filled with the region bounding boxes (ContainerType_Vector_TcVnRectangle_DINT; Non-zero interface pointers are reused.) *)
		hrPrev	:	HRESULT;	(* HRESULT indicating the result of previous operations (If SUCCEEDED(hrPrev) equals false, no operation is executed.) *)
	END_VAR

END_FUNCTION

// Functions/Keypoint Features/F_VN_RegionsMSERExp

	{attribute 'TcIecLibraryType'}
	{attribute 'external_name' := 'F_VN_RegionsMSERExp_GUID_88D0995E_EC24_43FD_D328_22E7CF7E8AF3'}
	(* Detects regions using the MSER method. (expert function) *)
	FUNCTION F_VN_RegionsMSERExp : HRESULT
	VAR_INPUT
		ipSrcImage	:	ITcVnImage;	(* Source image *)
		ipRegions	:	REFERENCE TO ITcVnContainer;	(* Returns a container which is filled with the region points (ContainerType_Vector_Vector_TcVnPoint2_DINT; Non-zero interface pointers are reused.) *)
		ipBoundingBoxes	:	REFERENCE TO ITcVnContainer;	(* Returns a container which is filled with the region bounding boxes (ContainerType_Vector_TcVnRectangle_DINT; Non-zero interface pointers are reused.) *)
	END_VAR
	VAR_IN_OUT
		stParams	:	TcVnParamsMSER;	(* Additional expert parameters *)
	END_VAR
	VAR_INPUT
		hrPrev	:	HRESULT;	(* HRESULT indicating the result of previous operations (If SUCCEEDED(hrPrev) equals false, no operation is executed.) *)
	END_VAR

END_FUNCTION

// Functions/Code Quality/F_VN_GradeBarcode

	{attribute 'TcIecLibraryType'}
	{attribute 'external_name' := 'F_VN_GradeBarcode_GUID_15BCE042_25A8_47E3_EE2F_2AE909E1A2F8'}
	(* Grades a 1D barcode according to ISO / IEC 15416:2016. Requires uniform illumination, good focus and the image sensor plane parallel to the code plane to achieve meaningful results. *)
	FUNCTION F_VN_GradeBarcode : HRESULT
	VAR_INPUT
		ipSrcImage	:	ITcVnImage;	(* Source image, only containing the horizontally aligned barcode region (USINT, 1 channel, including quiet zones on left and right, excluding Text or empty space on more than 10% total height on top or bottom) *)
		ipDecodedData	:	REFERENCE TO ITcVnContainer;	(* Returns the decoded data (ContainerType_String_SINT) *)
	END_VAR
	VAR_IN_OUT
		stCodeGrades	:	TcVnCodeGrades1D;	(* Returns the code grades in the range from 0 (very bad) to 4 (very good) *)
	END_VAR
	VAR_INPUT
		eBarcodeType	:	ETcVnBarcodeType;	(* Type of the barcode (supported: CODE39, CODE128, EAN8, EAN13, ITF, UPCA, UPCE) *)
		hrPrev	:	HRESULT;	(* HRESULT indicating the result of previous operations (If SUCCEEDED(hrPrev) equals false, no operation is executed.) *)
	END_VAR
	VAR_OUTPUT
		fAngleDeg	:	REAL;	(* Returns the approximate clockwise rotation angle in degree *)
	END_VAR

END_FUNCTION

// Functions/Code Quality/F_VN_GradeBarcodeExp

	{attribute 'TcIecLibraryType'}
	{attribute 'external_name' := 'F_VN_GradeBarcodeExp_GUID_9C6DAED7_BCF9_49C3_E364_D86CE1E53512'}
	(* Grades a 1D barcode according to ISO / IEC 15416:2016. Requires uniform illumination, good focus and the image sensor plane parallel to the code plane to achieve meaningful results. (expert function) *)
	FUNCTION F_VN_GradeBarcodeExp : HRESULT
	VAR_INPUT
		ipSrcImage	:	ITcVnImage;	(* Source image, only containing the horizontally aligned barcode region (USINT, 1 channel, including quiet zones on left and right, excluding Text or empty space on more than 10% total height on top or bottom) *)
		ipDecodedData	:	REFERENCE TO ITcVnContainer;	(* Returns the decoded data (ContainerType_String_SINT) *)
	END_VAR
	VAR_IN_OUT
		stCodeGrades	:	TcVnCodeGrades1D;	(* Returns the code grades in the range from 0 (very bad) to 4 (very good) *)
	END_VAR
	VAR_INPUT
		eBarcodeType	:	ETcVnBarcodeType;	(* Type of the barcode (supported: CODE39, CODE128, EAN8, EAN13, ITF, UPCA, UPCE) *)
		eSearchDirection	:	ETcVnBarcodeSearchDirection;	(* Barcode search direction (BSD_ANY first tries horizontal, then vertical) *)
		ipResultVisualization	:	REFERENCE TO ITcVnImage;	(* Returns a visualization of the scan lines (optional, set to 0 if not required). Grades are color coded: >= 3 as green, >= 2 as light blue, >= 1 as orange, < 1 as red *)
		ipScanLineInfo	:	REFERENCE TO ITcVnContainer;	(* Returns additional scan line info for further evaluation, e.g. to use PlotIntensityProfile for visualization (optional, set to 0 if not required; ContainerType_Vector_TcVnVector3_REAL, containing [row index, overall grade, threshold]) *)
		ipContour	:	REFERENCE TO ITcVnContainer;	(* Returns the 4 approximate code corner points, including the quiet zone (optional, set to 0 if not required; ContainerType_Vector_TcVnPoint2_DINT) *)
		hrPrev	:	HRESULT;	(* HRESULT indicating the result of previous operations (If SUCCEEDED(hrPrev) equals false, no operation is executed.) *)
	END_VAR
	VAR_OUTPUT
		fAngleDeg	:	REAL;	(* Returns the approximate clockwise rotation angle in degree *)
	END_VAR

END_FUNCTION

// Functions/Code Quality/F_VN_GradeDataMatrixCode

	{attribute 'TcIecLibraryType'}
	{attribute 'external_name' := 'F_VN_GradeDataMatrixCode_GUID_343B50E7_C52D_4495_E1B1_532C3DB47054'}
	(* Grades a Data Matrix code (ECC200) according to ISO / IEC 15415:2011. Requires uniform illumination, good focus and the image sensor plane parallel to the code plane to achieve meaningful results. *)
	FUNCTION F_VN_GradeDataMatrixCode : HRESULT
	VAR_INPUT
		ipSrcImage	:	ITcVnImage;	(* Source image, only containing the Data Matrix code region (USINT, 1 channel, including quiet zone) *)
		ipDecodedData	:	REFERENCE TO ITcVnContainer;	(* Returns the decoded data (ContainerType_String_SINT) *)
	END_VAR
	VAR_IN_OUT
		stCodeGrades	:	TcVnCodeGradesDM;	(* Returns the code grades in the range from 0 (very bad) to 4 (very good) *)
	END_VAR
	VAR_INPUT
		fModuleWidth	:	REAL;	(* Minimum module width of the code in the image (in pixels). Must be at least 3, preferably 5 - 8. *)
		hrPrev	:	HRESULT;	(* HRESULT indicating the result of previous operations (If SUCCEEDED(hrPrev) equals false, no operation is executed.) *)
	END_VAR
	VAR_OUTPUT
		fAngleDeg	:	REAL;	(* Returns the clockwise rotation angle in degree *)
	END_VAR

END_FUNCTION

// Functions/Code Quality/F_VN_GradeDataMatrixCodeExp

	{attribute 'TcIecLibraryType'}
	{attribute 'external_name' := 'F_VN_GradeDataMatrixCodeExp_GUID_D75964B2_9167_433B_DC2A_A3C354EB7686'}
	(* Grades a Data Matrix code (ECC200) according to ISO / IEC 15415:2011. Requires uniform illumination, good focus and the image sensor plane parallel to the code plane to achieve meaningful results. (expert function) *)
	FUNCTION F_VN_GradeDataMatrixCodeExp : HRESULT
	VAR_INPUT
		ipSrcImage	:	ITcVnImage;	(* Source image, only containing the Data Matrix code region (USINT, 1 channel, including quiet zone) *)
		ipDecodedData	:	REFERENCE TO ITcVnContainer;	(* Returns the decoded data (ContainerType_String_SINT) *)
	END_VAR
	VAR_IN_OUT
		stCodeGrades	:	TcVnCodeGradesDM;	(* Returns the code grades in the range from 0 (very bad) to 4 (very good) *)
	END_VAR
	VAR_INPUT
		fModuleWidth	:	REAL;	(* Minimum module width of the code in the image (in pixels). Must be at least 3, preferably 5 - 8. *)
		ipResultVisualization	:	REFERENCE TO ITcVnImage;	(* Returns a visualization of the scan grid (optional, set to 0 if not required). Module margin grades are color coded: >= 3 as green, >= 2 as light blue, >= 1 as orange, < 1 as red *)
		ipMarginGrades	:	REFERENCE TO ITcVnContainer;	(* Returns the individual margin grade for each module, e.g. to create a custom visualization (optional, set to 0 if not required; ContainerType_Vector_TcVnVector3_REAL, containing [x-position, y-position, grade]) *)
		ipContour	:	REFERENCE TO ITcVnContainer;	(* Returns the 4 code corner points, excluding the quiet zone (optional, set to 0 if not required; ContainerType_Vector_TcVnPoint2_DINT) *)
		hrPrev	:	HRESULT;	(* HRESULT indicating the result of previous operations (If SUCCEEDED(hrPrev) equals false, no operation is executed.) *)
	END_VAR
	VAR_OUTPUT
		fAngleDeg	:	REAL;	(* Returns the clockwise rotation angle in degree *)
	END_VAR

END_FUNCTION

// Functions/Code Quality/F_VN_GradeQRCode

	{attribute 'TcIecLibraryType'}
	{attribute 'external_name' := 'F_VN_GradeQRCode_GUID_B87BB656_B28F_4F95_EE47_B0BD88064FEC'}
	(* Grades a QR code according to ISO / IEC 15415:2011. Requires uniform illumination, good focus and the image sensor plane parallel to the code plane to achieve meaningful results. *)
	FUNCTION F_VN_GradeQRCode : HRESULT
	VAR_INPUT
		ipSrcImage	:	ITcVnImage;	(* Source image, only containing the QR code region (USINT, 1 channel, including quiet zone) *)
		ipDecodedData	:	REFERENCE TO ITcVnContainer;	(* Returns the decoded data (ContainerType_String_SINT) *)
	END_VAR
	VAR_IN_OUT
		stCodeGrades	:	TcVnCodeGradesQR;	(* Returns the code grades in the range from 0 (very bad) to 4 (very good) *)
	END_VAR
	VAR_INPUT
		fModuleWidth	:	REAL;	(* Minimum module width of the code in the image (in pixels). Must be at least 3, preferably 5 - 8. *)
		hrPrev	:	HRESULT;	(* HRESULT indicating the result of previous operations (If SUCCEEDED(hrPrev) equals false, no operation is executed.) *)
	END_VAR
	VAR_OUTPUT
		fAngleDeg	:	REAL;	(* Returns the clockwise rotation angle in degree *)
	END_VAR

END_FUNCTION

// Functions/Code Quality/F_VN_GradeQRCodeExp

	{attribute 'TcIecLibraryType'}
	{attribute 'external_name' := 'F_VN_GradeQRCodeExp_GUID_EB637094_C5AD_488D_C146_599B106C186E'}
	(* Grades a QR code according to ISO / IEC 15415:2011. Requires uniform illumination, good focus and the image sensor plane parallel to the code plane to achieve meaningful results. (expert function) *)
	FUNCTION F_VN_GradeQRCodeExp : HRESULT
	VAR_INPUT
		ipSrcImage	:	ITcVnImage;	(* Source image, only containing the QR code region (USINT, 1 channel, including quiet zone) *)
		ipDecodedData	:	REFERENCE TO ITcVnContainer;	(* Returns the decoded data (ContainerType_String_SINT) *)
	END_VAR
	VAR_IN_OUT
		stCodeGrades	:	TcVnCodeGradesQR;	(* Returns the code grades in the range from 0 (very bad) to 4 (very good) *)
	END_VAR
	VAR_INPUT
		fModuleWidth	:	REAL;	(* Minimum module width of the code in the image (in pixels). Must be at least 3, preferably 5 - 8. *)
		ipResultVisualization	:	REFERENCE TO ITcVnImage;	(* Returns a visualization of the scan grid (optional, set to 0 if not required). Module margin grades are color coded: >= 3 as green, >= 2 as light blue, >= 1 as orange, < 1 as red *)
		ipMarginGrades	:	REFERENCE TO ITcVnContainer;	(* Returns the individual margin grade for each module, e.g. to create a custom visualization (optional, set to 0 if not required; ContainerType_Vector_TcVnVector3_REAL, containing [x-position, y-position, grade]) *)
		ipContour	:	REFERENCE TO ITcVnContainer;	(* Returns the 4 code corner points, excluding the quiet zone (optional, set to 0 if not required; ContainerType_Vector_TcVnPoint2_DINT) *)
		hrPrev	:	HRESULT;	(* HRESULT indicating the result of previous operations (If SUCCEEDED(hrPrev) equals false, no operation is executed.) *)
	END_VAR
	VAR_OUTPUT
		fAngleDeg	:	REAL;	(* Returns the clockwise rotation angle in degree *)
	END_VAR

END_FUNCTION

// Functions/Texture Analysis/F_VN_Granulometry

	{attribute 'TcIecLibraryType'}
	{attribute 'external_name' := 'F_VN_Granulometry_GUID_72A1445E_6915_4710_FA72_82B95575C864'}
	(* Computes the granulometry of a textured image using morphological operations. *)
	FUNCTION F_VN_Granulometry : HRESULT
	VAR_INPUT
		ipImage	:	ITcVnImage;	(* Source image (1 channel) *)
		ipIntensityDiffs	:	REFERENCE TO ITcVnContainer;	(* Returns the intensity differences between successive structuring element sizes (CTcVnContainer_Vector_LREAL), which can be used as features for texture description. *)
		eMorphType	:	ETcVnMorphologicalOperator;	(* Only opening or closing are supported. *)
		nMinSize	:	UDINT;	(* Min structuring element size (odd, >= 3) *)
		nMaxSize	:	UDINT;	(* Max structuring element size (>= nMinSize) *)
		nStep	:	UDINT;	(* Step, by which nMinSize is incremented until nMaxSize is exceeded (even, >= 2). *)
		hrPrev	:	HRESULT;	(* HRESULT indicating the result of previous operations (If SUCCEEDED(hrPrev) equals false, no operation is executed.) *)
	END_VAR

END_FUNCTION

// Functions/Texture Analysis/F_VN_HaralickFeatures

	{attribute 'TcIecLibraryType'}
	{attribute 'external_name' := 'F_VN_HaralickFeatures_GUID_5FA621A8_1123_4082_DF67_A513AC539CA0'}
	(* Computes the Haralick features of a graylevel image, which describe the texture. *)
	FUNCTION F_VN_HaralickFeatures : HRESULT
	VAR_INPUT
		ipImage	:	ITcVnImage;	(* Source image (1 channel, USINT) *)
		ipFeatures	:	REFERENCE TO ITcVnContainer;	(* Returns the computed Haralick features (CTcVnContainer_Vector_LREAL). The returned feature set contains the mean and standard deviation for each of the first 13 Haralick features, computed for 0, 45, 90, 135 degrees. So there will be 26 features in total (f1 mean, f1 stdDev, f2 mean, f2 stdDev, ..., f13 mean, f13 stdDev). *)
		nDist	:	UDINT;	(* Distance *)
		hrPrev	:	HRESULT;	(* HRESULT indicating the result of previous operations (If SUCCEEDED(hrPrev) equals false, no operation is executed.) *)
	END_VAR

END_FUNCTION

// Functions/OCR/F_VN_OCR

	{attribute 'TcIecLibraryType'}
	{attribute 'external_name' := 'F_VN_OCR_GUID_D9A4CE6A_DBF6_4747_E040_5BCB34240814'}
	(* Detects and recognizes characters in a binary image (white characters on black background). *)
	FUNCTION F_VN_OCR : HRESULT
	VAR_INPUT
		ipSrcImage	:	ITcVnImage;	(* Source image (USINT, 1 channel, binary) *)
		eModel	:	ULINT;	(* Selection of OCR model types (ETcVnOcrModelType) *)
		ipCharacters	:	REFERENCE TO ITcVnContainer;	(* Returns the recognized characters (ContainerType_Vector_String_SINT) *)
		hrPrev	:	HRESULT;	(* HRESULT indicating the result of previous operations (If SUCCEEDED(hrPrev) equals false, no operation is executed.) *)
	END_VAR

END_FUNCTION

// Functions/OCR/F_VN_OCRExp

	{attribute 'TcIecLibraryType'}
	{attribute 'external_name' := 'F_VN_OCRExp_GUID_7251E972_3C73_4691_C26A_2644B61A93B0'}
	(* Detects and recognizes characters in a binary image (white characters on black background). (expert function) *)
	FUNCTION F_VN_OCRExp : HRESULT
	VAR_INPUT
		ipSrcImage	:	ITcVnImage;	(* Source image (USINT, 1 channel, binary) *)
		eModel	:	ULINT;	(* Selection of OCR model types (ETcVnOcrModelType) *)
		ipCharacters	:	REFERENCE TO ITcVnContainer;	(* Returns the recognized characters (ContainerType_Vector_String_SINT) *)
	END_VAR
	VAR_IN_OUT CONSTANT
		sPattern	:	STRING;	(* String pattern containing the format in which characters are presented *)
	END_VAR
	VAR_INPUT
		eOcrOptions	:	UDINT;	(* Specifies which options must be applied to the function (ETcVnOcrOptions) *)
		ipBoundingBoxes	:	REFERENCE TO ITcVnContainer;	(* Returns the corresponding bounding boxes of the recognized characters (ContainerType_Vector_TcVnRectangle_DINT, optional, set to 0 if not required) *)
		ipConfidences	:	REFERENCE TO ITcVnContainer;	(* Returns the corresponding classification confidences of the recognized characters (ContainerType_Vector_REAL, optional, set to 0 if not required) *)
		hrPrev	:	HRESULT;	(* HRESULT indicating the result of previous operations (If SUCCEEDED(hrPrev) equals false, no operation is executed.) *)
	END_VAR
	VAR_OUTPUT
		fMinConfidence	:	REAL;	(* Returns the minimum value of the confidences *)
	END_VAR

END_FUNCTION

// Functions/Code Reading/F_VN_ReadBarcode

	{attribute 'TcIecLibraryType'}
	{attribute 'external_name' := 'F_VN_ReadBarcode_GUID_12B8ED38_0744_4D53_CDD6_11586A04ED49'}
	(* Detect and interpret a 1d barcode within the provided image.
          Can be canceled by Watchdog. *)
	FUNCTION F_VN_ReadBarcode : HRESULT
	VAR_INPUT
		ipSrcImage	:	ITcVnImage;	(* Source image (USINT elements, 1 channel or 3 channel (3 channel input is expected to be RGB and internally converted to Gray)) *)
		ipDecodedData	:	REFERENCE TO ITcVnContainer;	(* Returns the decoded code (ContainerType_Vector_String_SINT) *)
		eBarcodeType	:	UDINT;	(* Types of barcode to search for (ETcVnBarcodeType) *)
		hrPrev	:	HRESULT;	(* HRESULT indicating the result of previous operations (If SUCCEEDED(hrPrev) equals false, no operation is executed.) *)
	END_VAR

END_FUNCTION

// Functions/Code Reading/F_VN_ReadBarcodeExp

	{attribute 'TcIecLibraryType'}
	{attribute 'external_name' := 'F_VN_ReadBarcodeExp_GUID_18367B83_16DB_476F_FF23_DA9E4075D3FA'}
	(* Detect and interpret a 1d barcode within the provided image.
          Can be canceled by Watchdog. *)
	FUNCTION F_VN_ReadBarcodeExp : HRESULT
	VAR_INPUT
		ipSrcImage	:	ITcVnImage;	(* Source image (USINT elements, 1 channel or 3 channel (3 channel input is expected to be RGB and internally converted to Gray)) *)
		ipDecodedData	:	REFERENCE TO ITcVnContainer;	(* Returns the decoded code (ContainerType_Vector_String_SINT) *)
		ipContours	:	REFERENCE TO ITcVnContainer;	(* Returns the code positions as contours (optional, set to 0 if not required; ContainerType_Vector_Vector_TcVnPoint2_DINT) *)
		eBarcodeType	:	UDINT;	(* Types of barcode to search for (ETcVnBarcodeType) *)
		nCodeNumber	:	DINT;	(* Number of 1d barcode that should be detected within the provided image (currently only 1 supported). *)
		eSearchDirection	:	ETcVnBarcodeSearchDirection;	(* Barcode search direction. *)
		hrPrev	:	HRESULT;	(* HRESULT indicating the result of previous operations (If SUCCEEDED(hrPrev) equals false, no operation is executed.) *)
	END_VAR

END_FUNCTION

// Functions/Code Reading/F_VN_ReadBarcodeExp2

	{attribute 'TcIecLibraryType'}
	{attribute 'external_name' := 'F_VN_ReadBarcodeExp2_GUID_D9F531F4_D252_4192_D41D_8D60F3EBDA2D'}
	(* Detect and interpret a 1d barcode within the provided image.
          Can be canceled by Watchdog. *)
	FUNCTION F_VN_ReadBarcodeExp2 : HRESULT
	VAR_INPUT
		ipSrcImage	:	ITcVnImage;	(* Source image (USINT elements, 1 channel or 3 channel (3 channel input is expected to be RGB and internally converted to Gray)) *)
		ipDecodedData	:	REFERENCE TO ITcVnContainer;	(* Returns the decoded code (ContainerType_Vector_String_SINT) *)
		ipContours	:	REFERENCE TO ITcVnContainer;	(* Returns the code positions as contours (optional, set to 0 if not required; ContainerType_Vector_Vector_TcVnPoint2_DINT) *)
		eBarcodeType	:	UDINT;	(* Types of barcode to search for (ETcVnBarcodeType) *)
		nCodeNumber	:	DINT;	(* Number of 1d barcode that should be detected within the provided image (currently only 1 supported). *)
		eSearchDirection	:	ETcVnBarcodeSearchDirection;	(* Barcode search direction. *)
		ipAngles	:	REFERENCE TO ITcVnContainer;	(* Returns the clockwise code rotation angles (optional, set to 0 if not required; ContainerType_Vector_REAL) *)
		hrPrev	:	HRESULT;	(* HRESULT indicating the result of previous operations (If SUCCEEDED(hrPrev) equals false, no operation is executed.) *)
	END_VAR

END_FUNCTION

// Functions/Code Reading/F_VN_ReadDataMatrixCode

	{attribute 'TcIecLibraryType'}
	{attribute 'external_name' := 'F_VN_ReadDataMatrixCode_GUID_D809F1EB_E5A9_4547_EEAF_6C7A25AE08EA'}
	(* Detect and interpret a data matrix code (ECC200) within the provided image. *)
	FUNCTION F_VN_ReadDataMatrixCode : HRESULT
	VAR_INPUT
		ipSrcImage	:	ITcVnImage;	(* Source image (USINT elements, 1 or 3 channels) *)
		ipDecodedData	:	REFERENCE TO ITcVnContainer;	(* Returns the decoded code (ContainerType_Vector_String_SINT) *)
		hrPrev	:	HRESULT;	(* HRESULT indicating the result of previous operations (If SUCCEEDED(hrPrev) equals false, no operation is executed.) *)
	END_VAR

END_FUNCTION

// Functions/Code Reading/F_VN_ReadDataMatrixCodeExp

	{attribute 'TcIecLibraryType'}
	{attribute 'external_name' := 'F_VN_ReadDataMatrixCodeExp_GUID_4652012D_CD62_4A2E_C6C7_AE6837D5C852'}
	(* Detect and interpret a data matrix code (ECC200) within the provided image. *)
	FUNCTION F_VN_ReadDataMatrixCodeExp : HRESULT
	VAR_INPUT
		ipSrcImage	:	ITcVnImage;	(* Source image (USINT elements, 1 or 3 channels) *)
		ipDecodedData	:	REFERENCE TO ITcVnContainer;	(* Returns the decoded code (ContainerType_Vector_String_SINT) *)
		ipContours	:	REFERENCE TO ITcVnContainer;	(* Returns the code positions as contours (optional, set to 0 if not required; ContainerType_Vector_Vector_TcVnPoint2_DINT) *)
		nCodeNumber	:	DINT;	(* Number of data matrix codes that should be detected within the provided image. (If set to -1, it tries to detect all data matrix codes.) *)
		eSearchStrategy	:	UDINT;	(* Used search strategy (ETcVn2dCodeSearchStrategy) *)
		hrPrev	:	HRESULT;	(* HRESULT indicating the result of previous operations (If SUCCEEDED(hrPrev) equals false, no operation is executed.) *)
	END_VAR

END_FUNCTION

// Functions/Code Reading/F_VN_ReadDataMatrixCodeExp2

	{attribute 'TcIecLibraryType'}
	{attribute 'external_name' := 'F_VN_ReadDataMatrixCodeExp2_GUID_96ED4AC1_6CC6_47F3_CDC3_AD142C1D6D2D'}
	(* Detect and interpret a data matrix code (ECC200) within the provided image. *)
	FUNCTION F_VN_ReadDataMatrixCodeExp2 : HRESULT
	VAR_INPUT
		ipSrcImage	:	ITcVnImage;	(* Source image (USINT elements, 1 or 3 channels) *)
		ipDecodedData	:	REFERENCE TO ITcVnContainer;	(* Returns the decoded code (ContainerType_Vector_String_SINT) *)
		ipContours	:	REFERENCE TO ITcVnContainer;	(* Returns the code positions as contours (optional, set to 0 if not required; ContainerType_Vector_Vector_TcVnPoint2_DINT) *)
		nCodeNumber	:	DINT;	(* Number of data matrix codes that should be detected within the provided image. (If set to -1, it tries to detect all data matrix codes.) *)
		eSearchStrategy	:	UDINT;	(* Used search strategy (ETcVn2dCodeSearchStrategy) *)
		ipAngles	:	REFERENCE TO ITcVnContainer;	(* Returns the clockwise code rotation angles (optional, set to 0 if not required; ContainerType_Vector_REAL) *)
		hrPrev	:	HRESULT;	(* HRESULT indicating the result of previous operations (If SUCCEEDED(hrPrev) equals false, no operation is executed.) *)
	END_VAR

END_FUNCTION

// Functions/Code Reading/F_VN_ReadPharmaCode

	{attribute 'TcIecLibraryType'}
	{attribute 'external_name' := 'F_VN_ReadPharmaCode_GUID_8ABFB2DF_8043_48F5_C88A_B4D9913461BE'}
	(* Detect and interpret a pharma code within the provided image.
				Can be canceled by Watchdog. *)
	FUNCTION F_VN_ReadPharmaCode : HRESULT
	VAR_INPUT
		ipSrcImage	:	ITcVnImage;	(* Source image (1 channel (all element types) or 3 channel with elements of type TCVN_ET_USINT, TCVN_ET_UINT or TCVN_ET_REAL (3 channel input is expected to be RGB and internally converted to Gray)) *)
		ipDecodedData	:	REFERENCE TO ITcVnContainer;	(* Returns the decoded code (ContainerType_Vector_String_SINT) *)
		hrPrev	:	HRESULT;	(* HRESULT indicating the result of previous operations (If SUCCEEDED(hrPrev) equals false, no operation is executed.) *)
	END_VAR

END_FUNCTION

// Functions/Code Reading/F_VN_ReadPharmaCodeExp

	{attribute 'TcIecLibraryType'}
	{attribute 'external_name' := 'F_VN_ReadPharmaCodeExp_GUID_8FA197FC_5937_4FF6_C737_D8C8869267F5'}
	(* Detect and interpret a pharma code within the provided image.
				Can be canceled by Watchdog. *)
	FUNCTION F_VN_ReadPharmaCodeExp : HRESULT
	VAR_INPUT
		ipSrcImage	:	ITcVnImage;	(* Source image (1 channel (all element types) or 3 channel with elements of type TCVN_ET_USINT, TCVN_ET_UINT or TCVN_ET_REAL (3 channel input is expected to be RGB and internally converted to Gray)) *)
		ipDecodedData	:	REFERENCE TO ITcVnContainer;	(* Returns the decoded code (ContainerType_Vector_String_SINT) *)
		ipContours	:	REFERENCE TO ITcVnContainer;	(* Returns the code positions as contours (optional, set to 0 if not required; ContainerType_Vector_Vector_TcVnPoint2_DINT) *)
		nCodeNumber	:	DINT;	(* Number of pharma codes that should be detected within the provided image (currently only 1 supported). *)
		nMinBarNumber	:	INT;	(* Minimal number of (dark) bars that codes must have. *)
		hrPrev	:	HRESULT;	(* HRESULT indicating the result of previous operations (If SUCCEEDED(hrPrev) equals false, no operation is executed.) *)
	END_VAR

END_FUNCTION

// Functions/Code Reading/F_VN_ReadPharmaCodeExp2

	{attribute 'TcIecLibraryType'}
	{attribute 'external_name' := 'F_VN_ReadPharmaCodeExp2_GUID_096DE644_38E7_45FA_F688_614F02BB219B'}
	(* Detect and interpret a pharma code within the provided image.
				Can be canceled by Watchdog. *)
	FUNCTION F_VN_ReadPharmaCodeExp2 : HRESULT
	VAR_INPUT
		ipSrcImage	:	ITcVnImage;	(* Source image (1 channel (all element types) or 3 channel with elements of type TCVN_ET_USINT, TCVN_ET_UINT or TCVN_ET_REAL (3 channel input is expected to be RGB and internally converted to Gray)) *)
		ipDecodedData	:	REFERENCE TO ITcVnContainer;	(* Returns the decoded code (ContainerType_Vector_String_SINT) *)
		ipContours	:	REFERENCE TO ITcVnContainer;	(* Returns the code positions as contours (optional, set to 0 if not required; ContainerType_Vector_Vector_TcVnPoint2_DINT) *)
		nCodeNumber	:	DINT;	(* Number of pharma codes that should be detected within the provided image (currently only 1 supported). *)
		nMinBarNumber	:	INT;	(* Minimal number of (dark) bars that codes must have. *)
		ipAngles	:	REFERENCE TO ITcVnContainer;	(* Returns the clockwise code rotation angles (optional, set to 0 if not required; ContainerType_Vector_REAL) *)
		hrPrev	:	HRESULT;	(* HRESULT indicating the result of previous operations (If SUCCEEDED(hrPrev) equals false, no operation is executed.) *)
	END_VAR

END_FUNCTION

// Functions/Code Reading/F_VN_ReadQRCode

	{attribute 'TcIecLibraryType'}
	{attribute 'external_name' := 'F_VN_ReadQRCode_GUID_0DE0D02A_926B_4335_E350_67B4926D0C7C'}
	(* Detect and interpret a QR code within the provided image.
          Can be canceled by Watchdog. *)
	FUNCTION F_VN_ReadQRCode : HRESULT
	VAR_INPUT
		ipSrcImage	:	ITcVnImage;	(* Source image (USINT elements, 1 channel or 3 channel (3 channel input is expected to be RGB and internally converted to Gray)) *)
		ipDecodedData	:	REFERENCE TO ITcVnContainer;	(* Returns the decoded code (ContainerType_Vector_String_SINT) *)
		hrPrev	:	HRESULT;	(* HRESULT indicating the result of previous operations (If SUCCEEDED(hrPrev) equals false, no operation is executed.) *)
	END_VAR

END_FUNCTION

// Functions/Code Reading/F_VN_ReadQRCodeExp

	{attribute 'TcIecLibraryType'}
	{attribute 'external_name' := 'F_VN_ReadQRCodeExp_GUID_80502B8F_8F4D_450C_E83D_3C621681D52E'}
	(* Detect and interpret a QR code within the provided image.
          Can be canceled by Watchdog. *)
	FUNCTION F_VN_ReadQRCodeExp : HRESULT
	VAR_INPUT
		ipSrcImage	:	ITcVnImage;	(* Source image (USINT elements, 1 channel or 3 channel (3 channel input is expected to be RGB and internally converted to Gray)) *)
		ipDecodedData	:	REFERENCE TO ITcVnContainer;	(* Returns the decoded code (ContainerType_Vector_String_SINT) *)
		ipContours	:	REFERENCE TO ITcVnContainer;	(* Returns the code positions as contours (optional, set to 0 if not required; ContainerType_Vector_Vector_TcVnPoint2_DINT) *)
		nCodeNumber	:	DINT;	(* Number of QR codes that should be detected within the provided image (currently only 1 supported). *)
		eSearchStrategy	:	UDINT;	(* Used search strategy (ETcVn2dCodeSearchStrategy) *)
		hrPrev	:	HRESULT;	(* HRESULT indicating the result of previous operations (If SUCCEEDED(hrPrev) equals false, no operation is executed.) *)
	END_VAR

END_FUNCTION

// Functions/Code Reading/F_VN_ReadQRCodeExp2

	{attribute 'TcIecLibraryType'}
	{attribute 'external_name' := 'F_VN_ReadQRCodeExp2_GUID_A5587F4A_A515_4E8A_D408_01ECA3FD7274'}
	(* Detect and interpret a QR code within the provided image.
          Can be canceled by Watchdog. *)
	FUNCTION F_VN_ReadQRCodeExp2 : HRESULT
	VAR_INPUT
		ipSrcImage	:	ITcVnImage;	(* Source image (USINT elements, 1 channel or 3 channel (3 channel input is expected to be RGB and internally converted to Gray)) *)
		ipDecodedData	:	REFERENCE TO ITcVnContainer;	(* Returns the decoded code (ContainerType_Vector_String_SINT) *)
		ipContours	:	REFERENCE TO ITcVnContainer;	(* Returns the code positions as contours (optional, set to 0 if not required; ContainerType_Vector_Vector_TcVnPoint2_DINT) *)
		nCodeNumber	:	DINT;	(* Number of QR codes that should be detected within the provided image (currently only 1 supported). *)
		eSearchStrategy	:	UDINT;	(* Used search strategy (ETcVn2dCodeSearchStrategy) *)
		ipAngles	:	REFERENCE TO ITcVnContainer;	(* Returns the clockwise code rotation angles (optional, set to 0 if not required; ContainerType_Vector_REAL) *)
		hrPrev	:	HRESULT;	(* HRESULT indicating the result of previous operations (If SUCCEEDED(hrPrev) equals false, no operation is executed.) *)
	END_VAR

END_FUNCTION

// Functions/Algebraic Container Operations/F_VN_AddToContainerElements/F_VN_AddToContainerElements_DINT

	{attribute 'TcIecLibraryType'}
	{attribute 'external_name' := 'F_VN_AddToContainerElements_DINT_GUID_ABDE051C_9CC0_4CA4_F9C5_BE076CF23598'}
	(* Add a value to each container element. *)
	FUNCTION F_VN_AddToContainerElements_DINT : HRESULT
	VAR_INPUT
		nValue	:	DINT;	(* Value *)
		ipContainer	:	ITcVnContainer;	(* Container with DINT elements *)
		hrPrev	:	HRESULT;	(* HRESULT indicating the result of previous operations (If SUCCEEDED(hrPrev) equals false, no operation is executed.) *)
	END_VAR

END_FUNCTION

// Functions/Algebraic Container Operations/F_VN_AddToContainerElements/F_VN_AddToContainerElements_INT

	{attribute 'TcIecLibraryType'}
	{attribute 'external_name' := 'F_VN_AddToContainerElements_INT_GUID_762BFCA9_9499_4E64_D388_0FF501168F3E'}
	(* Add a value to each container element. *)
	FUNCTION F_VN_AddToContainerElements_INT : HRESULT
	VAR_INPUT
		nValue	:	INT;	(* Value *)
		ipContainer	:	ITcVnContainer;	(* Container with INT elements *)
		hrPrev	:	HRESULT;	(* HRESULT indicating the result of previous operations (If SUCCEEDED(hrPrev) equals false, no operation is executed.) *)
	END_VAR

END_FUNCTION

// Functions/Algebraic Container Operations/F_VN_AddToContainerElements/F_VN_AddToContainerElements_LREAL

	{attribute 'TcIecLibraryType'}
	{attribute 'external_name' := 'F_VN_AddToContainerElements_LREAL_GUID_1457CF58_9C74_4ADF_C03E_63CF946B9414'}
	(* Add a value to each container element. *)
	FUNCTION F_VN_AddToContainerElements_LREAL : HRESULT
	VAR_INPUT
		fValue	:	LREAL;	(* Value *)
		ipContainer	:	ITcVnContainer;	(* Container with LREAL elements *)
		hrPrev	:	HRESULT;	(* HRESULT indicating the result of previous operations (If SUCCEEDED(hrPrev) equals false, no operation is executed.) *)
	END_VAR

END_FUNCTION

// Functions/Algebraic Container Operations/F_VN_AddToContainerElements/F_VN_AddToContainerElements_REAL

	{attribute 'TcIecLibraryType'}
	{attribute 'external_name' := 'F_VN_AddToContainerElements_REAL_GUID_996060AC_F7B5_40C2_D15B_861EBB4049D2'}
	(* Add a value to each container element. *)
	FUNCTION F_VN_AddToContainerElements_REAL : HRESULT
	VAR_INPUT
		fValue	:	REAL;	(* Value *)
		ipContainer	:	ITcVnContainer;	(* Container with REAL elements *)
		hrPrev	:	HRESULT;	(* HRESULT indicating the result of previous operations (If SUCCEEDED(hrPrev) equals false, no operation is executed.) *)
	END_VAR

END_FUNCTION

// Functions/Algebraic Container Operations/F_VN_AddToContainerElements/F_VN_AddToContainerElements_SINT

	{attribute 'TcIecLibraryType'}
	{attribute 'external_name' := 'F_VN_AddToContainerElements_SINT_GUID_D222E56E_CD69_44D6_D369_E19A3F5E193A'}
	(* Add a value to each container element. *)
	FUNCTION F_VN_AddToContainerElements_SINT : HRESULT
	VAR_INPUT
		nValue	:	SINT;	(* Value *)
		ipContainer	:	ITcVnContainer;	(* Container with SINT elements *)
		hrPrev	:	HRESULT;	(* HRESULT indicating the result of previous operations (If SUCCEEDED(hrPrev) equals false, no operation is executed.) *)
	END_VAR

END_FUNCTION

// Functions/Algebraic Container Operations/F_VN_AddToContainerElements/F_VN_AddToContainerElements_TcVnKeyPoint

	{attribute 'TcIecLibraryType'}
	{attribute 'external_name' := 'F_VN_AddToContainerElements_TcVnKeyPoint_GUID_CB126513_FF6D_446F_FE86_7BC84681EE12'}
	(* Add a value to each container element. *)
	FUNCTION F_VN_AddToContainerElements_TcVnKeyPoint : HRESULT
	VAR_IN_OUT
		stValue	:	TcVnKeyPoint;	(* Value *)
	END_VAR
	VAR_INPUT
		ipContainer	:	ITcVnContainer;	(* Container with TcVnKeyPoint elements *)
		hrPrev	:	HRESULT;	(* HRESULT indicating the result of previous operations (If SUCCEEDED(hrPrev) equals false, no operation is executed.) *)
	END_VAR

END_FUNCTION

// Functions/Algebraic Container Operations/F_VN_AddToContainerElements/F_VN_AddToContainerElements_TcVnPoint2_DINT

	{attribute 'TcIecLibraryType'}
	{attribute 'external_name' := 'F_VN_AddToContainerElements_TcVnPoint2_DINT_GUID_F1CE6D50_7C23_4732_CC2F_60EAEE70C164'}
	(* Add a value to each container element. *)
	FUNCTION F_VN_AddToContainerElements_TcVnPoint2_DINT : HRESULT
	VAR_IN_OUT
		aValue	:	TcVnPoint2_DINT;	(* Value *)
	END_VAR
	VAR_INPUT
		ipContainer	:	ITcVnContainer;	(* Container with TcVnPoint2_DINT elements *)
		hrPrev	:	HRESULT;	(* HRESULT indicating the result of previous operations (If SUCCEEDED(hrPrev) equals false, no operation is executed.) *)
	END_VAR

END_FUNCTION

// Functions/Algebraic Container Operations/F_VN_AddToContainerElements/F_VN_AddToContainerElements_TcVnPoint2_LREAL

	{attribute 'TcIecLibraryType'}
	{attribute 'external_name' := 'F_VN_AddToContainerElements_TcVnPoint2_LREAL_GUID_B33D351C_75D8_44E9_F273_FFD2AF5AFABF'}
	(* Add a value to each container element. *)
	FUNCTION F_VN_AddToContainerElements_TcVnPoint2_LREAL : HRESULT
	VAR_IN_OUT
		aValue	:	TcVnPoint2_LREAL;	(* Value *)
	END_VAR
	VAR_INPUT
		ipContainer	:	ITcVnContainer;	(* Container with TcVnPoint2_LREAL elements *)
		hrPrev	:	HRESULT;	(* HRESULT indicating the result of previous operations (If SUCCEEDED(hrPrev) equals false, no operation is executed.) *)
	END_VAR

END_FUNCTION

// Functions/Algebraic Container Operations/F_VN_AddToContainerElements/F_VN_AddToContainerElements_TcVnPoint2_REAL

	{attribute 'TcIecLibraryType'}
	{attribute 'external_name' := 'F_VN_AddToContainerElements_TcVnPoint2_REAL_GUID_F0DD7946_C505_4714_C568_EFA703F2826B'}
	(* Add a value to each container element. *)
	FUNCTION F_VN_AddToContainerElements_TcVnPoint2_REAL : HRESULT
	VAR_IN_OUT
		aValue	:	TcVnPoint2_REAL;	(* Value *)
	END_VAR
	VAR_INPUT
		ipContainer	:	ITcVnContainer;	(* Container with TcVnPoint2_REAL elements *)
		hrPrev	:	HRESULT;	(* HRESULT indicating the result of previous operations (If SUCCEEDED(hrPrev) equals false, no operation is executed.) *)
	END_VAR

END_FUNCTION

// Functions/Algebraic Container Operations/F_VN_AddToContainerElements/F_VN_AddToContainerElements_TcVnPoint3_LREAL

	{attribute 'TcIecLibraryType'}
	{attribute 'external_name' := 'F_VN_AddToContainerElements_TcVnPoint3_LREAL_GUID_73D08337_A7BD_4B19_E78F_0B66AB1F0C6C'}
	(* Add a value to each container element. *)
	FUNCTION F_VN_AddToContainerElements_TcVnPoint3_LREAL : HRESULT
	VAR_IN_OUT
		aValue	:	TcVnPoint3_LREAL;	(* Value *)
	END_VAR
	VAR_INPUT
		ipContainer	:	ITcVnContainer;	(* Container with TcVnPoint3_LREAL elements *)
		hrPrev	:	HRESULT;	(* HRESULT indicating the result of previous operations (If SUCCEEDED(hrPrev) equals false, no operation is executed.) *)
	END_VAR

END_FUNCTION

// Functions/Algebraic Container Operations/F_VN_AddToContainerElements/F_VN_AddToContainerElements_TcVnPoint3_REAL

	{attribute 'TcIecLibraryType'}
	{attribute 'external_name' := 'F_VN_AddToContainerElements_TcVnPoint3_REAL_GUID_8FCD4858_8B37_4914_D1E9_674BCA18C421'}
	(* Add a value to each container element. *)
	FUNCTION F_VN_AddToContainerElements_TcVnPoint3_REAL : HRESULT
	VAR_IN_OUT
		aValue	:	TcVnPoint3_REAL;	(* Value *)
	END_VAR
	VAR_INPUT
		ipContainer	:	ITcVnContainer;	(* Container with TcVnPoint3_REAL elements *)
		hrPrev	:	HRESULT;	(* HRESULT indicating the result of previous operations (If SUCCEEDED(hrPrev) equals false, no operation is executed.) *)
	END_VAR

END_FUNCTION

// Functions/Algebraic Container Operations/F_VN_AddToContainerElements/F_VN_AddToContainerElements_TcVnRectangle_DINT

	{attribute 'TcIecLibraryType'}
	{attribute 'external_name' := 'F_VN_AddToContainerElements_TcVnRectangle_DINT_GUID_A71FCEA4_9756_48ED_D843_A4DF29E91185'}
	(* Add a value to each container element. *)
	FUNCTION F_VN_AddToContainerElements_TcVnRectangle_DINT : HRESULT
	VAR_IN_OUT
		stValue	:	TcVnRectangle_DINT;	(* Value *)
	END_VAR
	VAR_INPUT
		ipContainer	:	ITcVnContainer;	(* Container with TcVnRectangle_DINT elements *)
		hrPrev	:	HRESULT;	(* HRESULT indicating the result of previous operations (If SUCCEEDED(hrPrev) equals false, no operation is executed.) *)
	END_VAR

END_FUNCTION

// Functions/Algebraic Container Operations/F_VN_AddToContainerElements/F_VN_AddToContainerElements_TcVnVector2_DINT

	{attribute 'TcIecLibraryType'}
	{attribute 'external_name' := 'F_VN_AddToContainerElements_TcVnVector2_DINT_GUID_0D480D9A_6C34_4CBF_F107_ADD9EF5DD131'}
	(* Add a value to each container element. *)
	FUNCTION F_VN_AddToContainerElements_TcVnVector2_DINT : HRESULT
	VAR_IN_OUT
		aValue	:	TcVnVector2_DINT;	(* Value *)
	END_VAR
	VAR_INPUT
		ipContainer	:	ITcVnContainer;	(* Container with TcVnVector2_DINT elements *)
		hrPrev	:	HRESULT;	(* HRESULT indicating the result of previous operations (If SUCCEEDED(hrPrev) equals false, no operation is executed.) *)
	END_VAR

END_FUNCTION

// Functions/Algebraic Container Operations/F_VN_AddToContainerElements/F_VN_AddToContainerElements_TcVnVector2_INT

	{attribute 'TcIecLibraryType'}
	{attribute 'external_name' := 'F_VN_AddToContainerElements_TcVnVector2_INT_GUID_AA3477AA_E8E6_42DA_D9CC_97BB0589CAEC'}
	(* Add a value to each container element. *)
	FUNCTION F_VN_AddToContainerElements_TcVnVector2_INT : HRESULT
	VAR_IN_OUT
		aValue	:	TcVnVector2_INT;	(* Value *)
	END_VAR
	VAR_INPUT
		ipContainer	:	ITcVnContainer;	(* Container with TcVnVector2_INT elements *)
		hrPrev	:	HRESULT;	(* HRESULT indicating the result of previous operations (If SUCCEEDED(hrPrev) equals false, no operation is executed.) *)
	END_VAR

END_FUNCTION

// Functions/Algebraic Container Operations/F_VN_AddToContainerElements/F_VN_AddToContainerElements_TcVnVector2_REAL

	{attribute 'TcIecLibraryType'}
	{attribute 'external_name' := 'F_VN_AddToContainerElements_TcVnVector2_REAL_GUID_E83D7C4E_7EAF_401B_C99F_0E7A276E2D57'}
	(* Add a value to each container element. *)
	FUNCTION F_VN_AddToContainerElements_TcVnVector2_REAL : HRESULT
	VAR_IN_OUT
		aValue	:	TcVnVector2_REAL;	(* Value *)
	END_VAR
	VAR_INPUT
		ipContainer	:	ITcVnContainer;	(* Container with TcVnVector2_REAL elements *)
		hrPrev	:	HRESULT;	(* HRESULT indicating the result of previous operations (If SUCCEEDED(hrPrev) equals false, no operation is executed.) *)
	END_VAR

END_FUNCTION

// Functions/Algebraic Container Operations/F_VN_AddToContainerElements/F_VN_AddToContainerElements_TcVnVector2_SINT

	{attribute 'TcIecLibraryType'}
	{attribute 'external_name' := 'F_VN_AddToContainerElements_TcVnVector2_SINT_GUID_4ACB9C8A_2B61_4E56_E31E_7EBC5863A5FB'}
	(* Add a value to each container element. *)
	FUNCTION F_VN_AddToContainerElements_TcVnVector2_SINT : HRESULT
	VAR_IN_OUT
		aValue	:	TcVnVector2_SINT;	(* Value *)
	END_VAR
	VAR_INPUT
		ipContainer	:	ITcVnContainer;	(* Container with TcVnVector2_SINT elements *)
		hrPrev	:	HRESULT;	(* HRESULT indicating the result of previous operations (If SUCCEEDED(hrPrev) equals false, no operation is executed.) *)
	END_VAR

END_FUNCTION

// Functions/Algebraic Container Operations/F_VN_AddToContainerElements/F_VN_AddToContainerElements_TcVnVector2_UINT

	{attribute 'TcIecLibraryType'}
	{attribute 'external_name' := 'F_VN_AddToContainerElements_TcVnVector2_UINT_GUID_A6786771_C6A0_4ABB_CBB3_C85243A2821C'}
	(* Add a value to each container element. *)
	FUNCTION F_VN_AddToContainerElements_TcVnVector2_UINT : HRESULT
	VAR_IN_OUT
		aValue	:	TcVnVector2_UINT;	(* Value *)
	END_VAR
	VAR_INPUT
		ipContainer	:	ITcVnContainer;	(* Container with TcVnVector2_UINT elements *)
		hrPrev	:	HRESULT;	(* HRESULT indicating the result of previous operations (If SUCCEEDED(hrPrev) equals false, no operation is executed.) *)
	END_VAR

END_FUNCTION

// Functions/Algebraic Container Operations/F_VN_AddToContainerElements/F_VN_AddToContainerElements_TcVnVector2_USINT

	{attribute 'TcIecLibraryType'}
	{attribute 'external_name' := 'F_VN_AddToContainerElements_TcVnVector2_USINT_GUID_E9CDA437_E4D8_4833_D6F8_EBF42B1922EF'}
	(* Add a value to each container element. *)
	FUNCTION F_VN_AddToContainerElements_TcVnVector2_USINT : HRESULT
	VAR_IN_OUT
		aValue	:	TcVnVector2_USINT;	(* Value *)
	END_VAR
	VAR_INPUT
		ipContainer	:	ITcVnContainer;	(* Container with TcVnVector2_USINT elements *)
		hrPrev	:	HRESULT;	(* HRESULT indicating the result of previous operations (If SUCCEEDED(hrPrev) equals false, no operation is executed.) *)
	END_VAR

END_FUNCTION

// Functions/Algebraic Container Operations/F_VN_AddToContainerElements/F_VN_AddToContainerElements_TcVnVector3_INT

	{attribute 'TcIecLibraryType'}
	{attribute 'external_name' := 'F_VN_AddToContainerElements_TcVnVector3_INT_GUID_81912DE6_E557_4B20_D5BC_E2A01825CA1F'}
	(* Add a value to each container element. *)
	FUNCTION F_VN_AddToContainerElements_TcVnVector3_INT : HRESULT
	VAR_IN_OUT
		aValue	:	TcVnVector3_INT;	(* Value *)
	END_VAR
	VAR_INPUT
		ipContainer	:	ITcVnContainer;	(* Container with TcVnVector3_INT elements *)
		hrPrev	:	HRESULT;	(* HRESULT indicating the result of previous operations (If SUCCEEDED(hrPrev) equals false, no operation is executed.) *)
	END_VAR

END_FUNCTION

// Functions/Algebraic Container Operations/F_VN_AddToContainerElements/F_VN_AddToContainerElements_TcVnVector3_REAL

	{attribute 'TcIecLibraryType'}
	{attribute 'external_name' := 'F_VN_AddToContainerElements_TcVnVector3_REAL_GUID_F7E31E1B_6AA1_40D2_C0DF_6AC560CBA321'}
	(* Add a value to each container element. *)
	FUNCTION F_VN_AddToContainerElements_TcVnVector3_REAL : HRESULT
	VAR_IN_OUT
		aValue	:	TcVnVector3_REAL;	(* Value *)
	END_VAR
	VAR_INPUT
		ipContainer	:	ITcVnContainer;	(* Container with TcVnVector3_REAL elements *)
		hrPrev	:	HRESULT;	(* HRESULT indicating the result of previous operations (If SUCCEEDED(hrPrev) equals false, no operation is executed.) *)
	END_VAR

END_FUNCTION

// Functions/Algebraic Container Operations/F_VN_AddToContainerElements/F_VN_AddToContainerElements_TcVnVector3_SINT

	{attribute 'TcIecLibraryType'}
	{attribute 'external_name' := 'F_VN_AddToContainerElements_TcVnVector3_SINT_GUID_9B12A624_F7AA_40C1_FA35_53536953B7BF'}
	(* Add a value to each container element. *)
	FUNCTION F_VN_AddToContainerElements_TcVnVector3_SINT : HRESULT
	VAR_IN_OUT
		aValue	:	TcVnVector3_SINT;	(* Value *)
	END_VAR
	VAR_INPUT
		ipContainer	:	ITcVnContainer;	(* Container with TcVnVector3_SINT elements *)
		hrPrev	:	HRESULT;	(* HRESULT indicating the result of previous operations (If SUCCEEDED(hrPrev) equals false, no operation is executed.) *)
	END_VAR

END_FUNCTION

// Functions/Algebraic Container Operations/F_VN_AddToContainerElements/F_VN_AddToContainerElements_TcVnVector3_UINT

	{attribute 'TcIecLibraryType'}
	{attribute 'external_name' := 'F_VN_AddToContainerElements_TcVnVector3_UINT_GUID_327774A1_D287_4A23_CD1A_0474A51D818A'}
	(* Add a value to each container element. *)
	FUNCTION F_VN_AddToContainerElements_TcVnVector3_UINT : HRESULT
	VAR_IN_OUT
		aValue	:	TcVnVector3_UINT;	(* Value *)
	END_VAR
	VAR_INPUT
		ipContainer	:	ITcVnContainer;	(* Container with TcVnVector3_UINT elements *)
		hrPrev	:	HRESULT;	(* HRESULT indicating the result of previous operations (If SUCCEEDED(hrPrev) equals false, no operation is executed.) *)
	END_VAR

END_FUNCTION

// Functions/Algebraic Container Operations/F_VN_AddToContainerElements/F_VN_AddToContainerElements_TcVnVector3_USINT

	{attribute 'TcIecLibraryType'}
	{attribute 'external_name' := 'F_VN_AddToContainerElements_TcVnVector3_USINT_GUID_271F4B8A_1626_4677_CA8E_DBED624CEB48'}
	(* Add a value to each container element. *)
	FUNCTION F_VN_AddToContainerElements_TcVnVector3_USINT : HRESULT
	VAR_IN_OUT
		aValue	:	TcVnVector3_USINT;	(* Value *)
	END_VAR
	VAR_INPUT
		ipContainer	:	ITcVnContainer;	(* Container with TcVnVector3_USINT elements *)
		hrPrev	:	HRESULT;	(* HRESULT indicating the result of previous operations (If SUCCEEDED(hrPrev) equals false, no operation is executed.) *)
	END_VAR

END_FUNCTION

// Functions/Algebraic Container Operations/F_VN_AddToContainerElements/F_VN_AddToContainerElements_TcVnVector4_DINT

	{attribute 'TcIecLibraryType'}
	{attribute 'external_name' := 'F_VN_AddToContainerElements_TcVnVector4_DINT_GUID_270F9096_16AB_4894_D4EB_D36E77CB30A1'}
	(* Add a value to each container element. *)
	FUNCTION F_VN_AddToContainerElements_TcVnVector4_DINT : HRESULT
	VAR_IN_OUT
		aValue	:	TcVnVector4_DINT;	(* Value *)
	END_VAR
	VAR_INPUT
		ipContainer	:	ITcVnContainer;	(* Container with TcVnVector4_DINT elements *)
		hrPrev	:	HRESULT;	(* HRESULT indicating the result of previous operations (If SUCCEEDED(hrPrev) equals false, no operation is executed.) *)
	END_VAR

END_FUNCTION

// Functions/Algebraic Container Operations/F_VN_AddToContainerElements/F_VN_AddToContainerElements_TcVnVector4_INT

	{attribute 'TcIecLibraryType'}
	{attribute 'external_name' := 'F_VN_AddToContainerElements_TcVnVector4_INT_GUID_A7CE4A42_4F6C_448C_D311_D7BF2B80B1FA'}
	(* Add a value to each container element. *)
	FUNCTION F_VN_AddToContainerElements_TcVnVector4_INT : HRESULT
	VAR_IN_OUT
		aValue	:	TcVnVector4_INT;	(* Value *)
	END_VAR
	VAR_INPUT
		ipContainer	:	ITcVnContainer;	(* Container with TcVnVector4_INT elements *)
		hrPrev	:	HRESULT;	(* HRESULT indicating the result of previous operations (If SUCCEEDED(hrPrev) equals false, no operation is executed.) *)
	END_VAR

END_FUNCTION

// Functions/Algebraic Container Operations/F_VN_AddToContainerElements/F_VN_AddToContainerElements_TcVnVector4_LREAL

	{attribute 'TcIecLibraryType'}
	{attribute 'external_name' := 'F_VN_AddToContainerElements_TcVnVector4_LREAL_GUID_C6484FFA_6D8C_4050_E9B1_3B7D852DF6C2'}
	(* Add a value to each container element. *)
	FUNCTION F_VN_AddToContainerElements_TcVnVector4_LREAL : HRESULT
	VAR_IN_OUT
		aValue	:	TcVnVector4_LREAL;	(* Value *)
	END_VAR
	VAR_INPUT
		ipContainer	:	ITcVnContainer;	(* Container with TcVnVector4_LREAL elements *)
		hrPrev	:	HRESULT;	(* HRESULT indicating the result of previous operations (If SUCCEEDED(hrPrev) equals false, no operation is executed.) *)
	END_VAR

END_FUNCTION

// Functions/Algebraic Container Operations/F_VN_AddToContainerElements/F_VN_AddToContainerElements_TcVnVector4_SINT

	{attribute 'TcIecLibraryType'}
	{attribute 'external_name' := 'F_VN_AddToContainerElements_TcVnVector4_SINT_GUID_E86D9FAD_9989_4AC0_EE5B_C32F9EF3D976'}
	(* Add a value to each container element. *)
	FUNCTION F_VN_AddToContainerElements_TcVnVector4_SINT : HRESULT
	VAR_IN_OUT
		aValue	:	TcVnVector4_SINT;	(* Value *)
	END_VAR
	VAR_INPUT
		ipContainer	:	ITcVnContainer;	(* Container with TcVnVector4_SINT elements *)
		hrPrev	:	HRESULT;	(* HRESULT indicating the result of previous operations (If SUCCEEDED(hrPrev) equals false, no operation is executed.) *)
	END_VAR

END_FUNCTION

// Functions/Algebraic Container Operations/F_VN_AddToContainerElements/F_VN_AddToContainerElements_TcVnVector4_UINT

	{attribute 'TcIecLibraryType'}
	{attribute 'external_name' := 'F_VN_AddToContainerElements_TcVnVector4_UINT_GUID_A1CA81B2_8FCE_4AC9_E438_A48CBC44091D'}
	(* Add a value to each container element. *)
	FUNCTION F_VN_AddToContainerElements_TcVnVector4_UINT : HRESULT
	VAR_IN_OUT
		aValue	:	TcVnVector4_UINT;	(* Value *)
	END_VAR
	VAR_INPUT
		ipContainer	:	ITcVnContainer;	(* Container with TcVnVector4_UINT elements *)
		hrPrev	:	HRESULT;	(* HRESULT indicating the result of previous operations (If SUCCEEDED(hrPrev) equals false, no operation is executed.) *)
	END_VAR

END_FUNCTION

// Functions/Algebraic Container Operations/F_VN_AddToContainerElements/F_VN_AddToContainerElements_TcVnVector4_USINT

	{attribute 'TcIecLibraryType'}
	{attribute 'external_name' := 'F_VN_AddToContainerElements_TcVnVector4_USINT_GUID_87152387_2528_437B_D036_20ABAABF9E5A'}
	(* Add a value to each container element. *)
	FUNCTION F_VN_AddToContainerElements_TcVnVector4_USINT : HRESULT
	VAR_IN_OUT
		aValue	:	TcVnVector4_USINT;	(* Value *)
	END_VAR
	VAR_INPUT
		ipContainer	:	ITcVnContainer;	(* Container with TcVnVector4_USINT elements *)
		hrPrev	:	HRESULT;	(* HRESULT indicating the result of previous operations (If SUCCEEDED(hrPrev) equals false, no operation is executed.) *)
	END_VAR

END_FUNCTION

// Functions/Algebraic Container Operations/F_VN_AddToContainerElements/F_VN_AddToContainerElements_UDINT

	{attribute 'TcIecLibraryType'}
	{attribute 'external_name' := 'F_VN_AddToContainerElements_UDINT_GUID_AE807CC7_EBFF_4932_FE6D_79818C344409'}
	(* Add a value to each container element. *)
	FUNCTION F_VN_AddToContainerElements_UDINT : HRESULT
	VAR_INPUT
		nValue	:	UDINT;	(* Value *)
		ipContainer	:	ITcVnContainer;	(* Container with UDINT elements *)
		hrPrev	:	HRESULT;	(* HRESULT indicating the result of previous operations (If SUCCEEDED(hrPrev) equals false, no operation is executed.) *)
	END_VAR

END_FUNCTION

// Functions/Algebraic Container Operations/F_VN_AddToContainerElements/F_VN_AddToContainerElements_UINT

	{attribute 'TcIecLibraryType'}
	{attribute 'external_name' := 'F_VN_AddToContainerElements_UINT_GUID_5A84E1C4_C182_4C0E_CD4C_368EF636CCD5'}
	(* Add a value to each container element. *)
	FUNCTION F_VN_AddToContainerElements_UINT : HRESULT
	VAR_INPUT
		nValue	:	UINT;	(* Value *)
		ipContainer	:	ITcVnContainer;	(* Container with UINT elements *)
		hrPrev	:	HRESULT;	(* HRESULT indicating the result of previous operations (If SUCCEEDED(hrPrev) equals false, no operation is executed.) *)
	END_VAR

END_FUNCTION

// Functions/Algebraic Container Operations/F_VN_AddToContainerElements/F_VN_AddToContainerElements_ULINT

	{attribute 'TcIecLibraryType'}
	{attribute 'external_name' := 'F_VN_AddToContainerElements_ULINT_GUID_75F2C5DB_7175_45F2_FDCC_117081AF54A8'}
	(* Add a value to each container element. *)
	FUNCTION F_VN_AddToContainerElements_ULINT : HRESULT
	VAR_INPUT
		nValue	:	ULINT;	(* Value *)
		ipContainer	:	ITcVnContainer;	(* Container with ULINT elements *)
		hrPrev	:	HRESULT;	(* HRESULT indicating the result of previous operations (If SUCCEEDED(hrPrev) equals false, no operation is executed.) *)
	END_VAR

END_FUNCTION

// Functions/Algebraic Container Operations/F_VN_AddToContainerElements/F_VN_AddToContainerElements_USINT

	{attribute 'TcIecLibraryType'}
	{attribute 'external_name' := 'F_VN_AddToContainerElements_USINT_GUID_ABBEC4E5_1E0F_4B04_D76C_5AF7359D2D4F'}
	(* Add a value to each container element. *)
	FUNCTION F_VN_AddToContainerElements_USINT : HRESULT
	VAR_INPUT
		nValue	:	USINT;	(* Value *)
		ipContainer	:	ITcVnContainer;	(* Container with USINT elements *)
		hrPrev	:	HRESULT;	(* HRESULT indicating the result of previous operations (If SUCCEEDED(hrPrev) equals false, no operation is executed.) *)
	END_VAR

END_FUNCTION

// Functions/Image Analysis/Object Detection/F_VN_AdjustActiveContour

	{attribute 'TcIecLibraryType'}
	{attribute 'external_name' := 'F_VN_AdjustActiveContour_GUID_18E5158B_69DF_434F_D839_B264A2455A75'}
	(* Adjust active contour (snake) in order to minimize its cummulative (internal and external) energy. *)
	FUNCTION F_VN_AdjustActiveContour : HRESULT
	VAR_INPUT
		ipImage	:	ITcVnImage;	(* Source image (1 channel, USINT elements) *)
		ipActiveContour	:	ITcVnContainer;	(* Initial contour, which will be adjusted *)
		fAlpha	:	REAL;	(* Continuity energy coefficient *)
		fBeta	:	REAL;	(* Curvature energy coefficient *)
		fGamma	:	REAL;	(* Image energy coefficient *)
		nWindowWidth	:	UDINT;	(* Window width (3, 5, 7, ...) *)
		nWindowHeight	:	UDINT;	(* Window height (3, 5, 7, ...) *)
		nMaxIterations	:	UDINT;	(* Maximum iterations *)
		bUseGradient	:	BOOL;	(* If true, the gradient magnitude is used as image energy (otherwise: pixel intensity) *)
		hrPrev	:	HRESULT;	(* HRESULT indicating the result of previous operations (If SUCCEEDED(hrPrev) equals false, no operation is executed.) *)
	END_VAR

END_FUNCTION

// Functions/Image Analysis/Object Detection/F_VN_DetectBlobs

	{attribute 'TcIecLibraryType'}
	{attribute 'external_name' := 'F_VN_DetectBlobs_GUID_2926A26C_03AC_43C6_E53B_64D65EAA331C'}
	(* Detects blob-contours. Applies a threshold, a contour search and offers several options for filtering the found contours. Provides easy setup for multiple thresholds and combination of results. *)
	FUNCTION F_VN_DetectBlobs : HRESULT
	VAR_INPUT
		ipSrcImage	:	ITcVnImage;	(* Source image (USINT or REAL, 1 channel or 3 channel (3 channel input is expected to be RGB and internally converted to Gray)) *)
		ipBlobContours	:	REFERENCE TO ITcVnContainer;	(* Returns a container which is filled with the found contours (ContainerType_Vector_Vector_TcVnPoint2_DINT; The elements of this container are single contours. Non-zero interface pointers are reused.) *)
	END_VAR
	VAR_IN_OUT
		stParams	:	TcVnParamsBlobDetection;	(* Parameters to filter the detected contours. *)
	END_VAR
	VAR_INPUT
		hrPrev	:	HRESULT;	(* HRESULT indicating the result of previous operations (If SUCCEEDED(hrPrev) equals false, no operation is executed.) *)
	END_VAR

END_FUNCTION

// Functions/Image Analysis/Object Detection/F_VN_DetectBlobsExp

	{attribute 'TcIecLibraryType'}
	{attribute 'external_name' := 'F_VN_DetectBlobsExp_GUID_0C5C0245_D5C7_4356_CF8C_B47851A141B6'}
	(* Detects blob-contours. Applies a threshold, a contour search and offers several options for filtering the found contours. Provides easy setup for multiple thresholds and combination of results. (expert function) *)
	FUNCTION F_VN_DetectBlobsExp : HRESULT
	VAR_INPUT
		ipSrcImage	:	ITcVnImage;	(* Source image (USINT or REAL, 1 channel or 3 channel (3 channel input is expected to be RGB and internally converted to Gray)) *)
		ipBlobContours	:	REFERENCE TO ITcVnContainer;	(* Returns a container which is filled with the found contours (ContainerType_Vector_Vector_TcVnPoint2_DINT; The elements of this container are single contours. Non-zero interface pointers are reused.) *)
	END_VAR
	VAR_IN_OUT
		stParams	:	TcVnParamsBlobDetection;	(* Parameters to filter the detected contours. *)
		aOffset	:	TcVnPoint;	(* Offset by which every contour point is shifted *)
	END_VAR
	VAR_INPUT
		hrPrev	:	HRESULT;	(* HRESULT indicating the result of previous operations (If SUCCEEDED(hrPrev) equals false, no operation is executed.) *)
	END_VAR

END_FUNCTION

// Functions/Image Analysis/Object Detection/F_VN_FindContourHierarchyExp

	{attribute 'TcIecLibraryType'}
	{attribute 'external_name' := 'F_VN_FindContourHierarchyExp_GUID_643E90CF_C41D_408B_CA02_238E7E7CB734'}
	(* Search for object contours in a binary image and determine their hierarchical relationship. (expert function) *)
	FUNCTION F_VN_FindContourHierarchyExp : HRESULT
	VAR_INPUT
		ipSrcImage	:	ITcVnImage;	(* Source image (1 channel, binary) *)
		ipContours	:	REFERENCE TO ITcVnContainer;	(* Returns a container which is filled with the found contours (ContainerType_Vector_Vector_TcVnPoint2_DINT; The elements of this container are single contours. Non-zero interface pointers are reused.) *)
		ipHierarchy	:	REFERENCE TO ITcVnContainer;	(* Returns a container which is filled with information on the found contours' hierarchy (ContainerType_Vector_TcVnVector4_DINT; The elements of this container are four-dimensional vectors containing the 0-based indices of the next [0] and the previous contour [1] at the same level, the first child [2], and the parent [3]. Non-zero interface pointers are reused.) *)
		eRetrievalMode	:	ETcVnContourRetrievalMode;	(* Specifies which contours are retrieved and how their relationship is encoded *)
		eApproximationMethod	:	ETcVnContourApproximationMethod;	(* Contour encoding *)
	END_VAR
	VAR_IN_OUT
		aOffset	:	TcVnPoint;	(* Offset by which every contour point is shifted *)
	END_VAR
	VAR_INPUT
		hrPrev	:	HRESULT;	(* HRESULT indicating the result of previous operations (If SUCCEEDED(hrPrev) equals false, no operation is executed.) *)
	END_VAR

END_FUNCTION

// Functions/Image Analysis/Object Detection/F_VN_FindContours

	{attribute 'TcIecLibraryType'}
	{attribute 'external_name' := 'F_VN_FindContours_GUID_0CF5BDB8_73E1_43B8_FC99_8BCA66834DC7'}
	(* Search for object contours in a binary image. Returns only external contours. *)
	FUNCTION F_VN_FindContours : HRESULT
	VAR_INPUT
		ipSrcImage	:	ITcVnImage;	(* Source image (1 channel, binary) *)
		ipContours	:	REFERENCE TO ITcVnContainer;	(* Returns a container which is filled with the found contours (ContainerType_Vector_Vector_TcVnPoint2_DINT; The elements of this container are single contours. Non-zero interface pointers are reused.) *)
		hrPrev	:	HRESULT;	(* HRESULT indicating the result of previous operations (If SUCCEEDED(hrPrev) equals false, no operation is executed.) *)
	END_VAR

END_FUNCTION

// Functions/Image Analysis/Object Detection/F_VN_FindContoursExp

	{attribute 'TcIecLibraryType'}
	{attribute 'external_name' := 'F_VN_FindContoursExp_GUID_7CF77E24_18BB_41AE_D882_7552EBFC75A9'}
	(* Search for object contours in a binary image. (expert function) *)
	FUNCTION F_VN_FindContoursExp : HRESULT
	VAR_INPUT
		ipSrcImage	:	ITcVnImage;	(* Source image (1 channel, binary) *)
		ipContours	:	REFERENCE TO ITcVnContainer;	(* Returns a container which is filled with the found contours (ContainerType_Vector_Vector_TcVnPoint2_DINT; The elements of this container are single contours. Non-zero interface pointers are reused.) *)
		eRetrievalMode	:	ETcVnContourRetrievalMode;	(* Specifies which contours are retrieved and how their relationship is encoded *)
		eApproximationMethod	:	ETcVnContourApproximationMethod;	(* Contour encoding *)
	END_VAR
	VAR_IN_OUT
		aOffset	:	TcVnPoint;	(* Offset by which every contour point is shifted *)
	END_VAR
	VAR_INPUT
		hrPrev	:	HRESULT;	(* HRESULT indicating the result of previous operations (If SUCCEEDED(hrPrev) equals false, no operation is executed.) *)
	END_VAR

END_FUNCTION

// Functions/Image Analysis/Object Detection/F_VN_HoughCircles

